C01822=1228.757,-113.151,-35.858,179.412,5.295,149.097
C01823=1228.752,-112.901,-35.869,179.414,5.294,149.096
C01824=1228.747,-112.651,-35.879,179.416,5.295,149.096
C01825=1228.741,-112.401,-35.889,179.418,5.294,149.095
C01826=1228.736,-112.152,-35.899,179.421,5.295,149.094
C01827=1228.731,-111.902,-35.910,179.423,5.295,149.094
C01828=1228.726,-111.652,-35.920,179.425,5.295,149.093
C01829=1228.720,-111.403,-35.930,179.427,5.295,149.092
C01830=1228.715,-111.153,-35.941,179.430,5.295,149.091
C01831=1228.710,-110.903,-35.950,179.432,5.295,149.091
C01832=1228.704,-110.653,-35.960,179.434,5.295,149.090
C01833=1228.699,-110.403,-35.970,179.437,5.295,149.089
C01834=1228.694,-110.153,-35.980,179.439,5.295,149.089
C01835=1228.688,-109.904,-35.991,179.442,5.295,149.088
C01836=1228.684,-109.655,-36.001,179.443,5.295,149.087
C01837=1228.679,-109.405,-36.012,179.446,5.296,149.087
C01838=1228.673,-109.156,-36.022,179.448,5.295,149.086
C01839=1228.668,-108.905,-36.032,179.451,5.296,149.085
C01840=1228.662,-108.656,-36.043,179.453,5.295,149.085
C01841=1228.657,-108.405,-36.053,179.456,5.296,149.084
C01842=1228.653,-108.156,-36.063,179.458,5.295,149.083
C01843=1228.647,-107.907,-36.073,179.460,5.296,149.082
C01844=1228.642,-107.656,-36.084,179.462,5.295,149.082
C01845=1228.636,-107.407,-36.094,179.465,5.296,149.081
C01846=1228.631,-107.157,-36.104,179.467,5.296,149.080
C01847=1228.626,-106.907,-36.115,179.469,5.295,149.080
C01848=1228.621,-106.658,-36.124,179.471,5.296,149.079
C01849=1228.616,-106.408,-36.135,179.474,5.296,149.078
C01850=1228.610,-106.158,-36.145,179.476,5.296,149.078
C01851=1228.606,-105.908,-36.156,179.478,5.296,149.077
C01852=1228.600,-105.659,-36.166,179.481,5.296,149.076
C01853=1228.595,-105.409,-36.177,179.483,5.296,149.075
C01854=1228.589,-105.159,-36.187,179.486,5.296,149.075
C01855=1228.584,-104.910,-36.197,179.488,5.296,149.074
C01856=1228.579,-104.659,-36.208,179.491,5.296,149.073
C01857=1228.574,-104.410,-36.218,179.492,5.296,149.073
C01858=1228.569,-104.160,-36.228,179.495,5.297,149.072
C01859=1228.564,-103.911,-36.239,179.497,5.296,149.071
C01860=1228.559,-103.661,-36.250,179.500,5.297,149.071
C01861=1228.553,-103.411,-36.260,179.502,5.296,149.070
C01862=1228.548,-103.161,-36.270,179.504,5.296,149.069
C01863=1228.542,-102.911,-36.281,179.506,5.296,149.069
C01864=1228.537,-102.662,-36.292,179.509,5.296,149.068
C01865=1228.532,-102.412,-36.302,179.511,5.296,149.067
C01866=1228.527,-102.163,-36.312,179.513,5.296,149.066
C01867=1228.522,-101.912,-36.323,179.516,5.297,149.066
C01868=1228.516,-101.663,-36.333,179.518,5.296,149.065
C01869=1228.511,-101.413,-36.344,179.521,5.297,149.064
C01870=1228.506,-101.164,-36.355,179.522,5.297,149.064
C01871=1228.501,-100.892,-36.366,179.526,5.297,149.063
C01872=1228.495,-100.621,-36.378,179.528,5.296,149.062
C01873=1228.489,-100.351,-36.388,179.530,5.297,149.061
C01874=1228.483,-100.080,-36.401,179.533,5.297,149.061
C01875=1228.478,-99.830,-36.411,179.535,5.297,149.060
C01876=1228.473,-99.580,-36.421,179.538,5.297,149.059
C01877=1228.468,-99.330,-36.433,179.540,5.297,149.059
C01878=1228.463,-99.081,-36.443,179.543,5.297,149.058
C01879=1228.458,-98.831,-36.454,179.545,5.297,149.057
C01880=1228.452,-98.581,-36.464,179.547,5.297,149.056
C01881=1228.447,-98.332,-36.475,179.549,5.297,149.056
C01882=1228.442,-98.082,-36.485,179.552,5.298,149.055
C01883=1228.437,-97.832,-36.496,179.554,5.297,149.054
C01884=1228.431,-97.583,-36.507,179.556,5.297,149.054
C01885=1228.426,-97.333,-36.517,179.558,5.298,149.053
C01886=1228.421,-97.083,-36.528,179.561,5.297,149.052
C01887=1228.416,-96.833,-36.539,179.563,5.298,149.052
C01888=1228.411,-96.584,-36.549,179.565,5.297,149.051
C01889=1228.406,-96.334,-36.560,179.568,5.298,149.050
C01890=1228.400,-96.084,-36.571,179.570,5.297,149.050
C01891=1228.395,-95.834,-36.582,179.573,5.298,149.049
C01892=1228.390,-95.584,-36.593,179.575,5.298,149.048
C01893=1228.384,-95.335,-36.603,179.578,5.298,149.047
C01894=1228.380,-95.085,-36.615,179.580,5.298,149.047
C01895=1228.374,-94.836,-36.625,179.582,5.298,149.046
C01896=1228.369,-94.586,-36.635,179.584,5.298,149.045
C01897=1228.364,-94.337,-36.646,179.587,5.298,149.045
C01898=1228.359,-94.086,-36.657,179.589,5.298,149.044
C01899=1228.353,-93.837,-36.668,179.592,5.298,149.043
C01900=1228.348,-93.587,-36.679,179.593,5.298,149.043
C01901=1228.343,-93.337,-36.690,179.596,5.299,149.042
C01902=1228.337,-93.088,-36.700,179.598,5.298,149.041
C01903=1228.333,-92.838,-36.712,179.601,5.299,149.041
C01904=1228.327,-92.589,-36.722,179.603,5.298,149.040
C01905=1228.322,-92.338,-36.732,179.606,5.299,149.039
C01906=1228.317,-92.089,-36.744,179.608,5.299,149.038
C01907=1228.311,-91.839,-36.755,179.610,5.299,149.038
C01908=1228.306,-91.589,-36.766,179.612,5.299,149.037
C01909=1228.301,-91.340,-36.776,179.615,5.299,149.036
C01910=1228.296,-91.090,-36.787,179.617,5.299,149.036
C01911=1228.291,-90.840,-36.799,179.620,5.299,149.035
C01912=1228.285,-90.591,-36.809,179.622,5.299,149.034
C01913=1228.280,-90.341,-36.821,179.625,5.299,149.033
C01914=1228.275,-90.091,-36.831,179.627,5.299,149.033
C01915=1228.270,-89.842,-36.842,179.629,5.299,149.032
C01916=1228.265,-89.592,-36.853,179.632,5.299,149.031
C01917=1228.259,-89.342,-36.864,179.634,5.299,149.031
C01918=1228.254,-89.092,-36.875,179.636,5.299,149.030
C01919=1228.249,-88.842,-36.886,179.639,5.299,149.029
C01920=1228.244,-88.593,-36.897,179.641,5.299,149.028
C01921=1228.239,-88.343,-36.908,179.643,5.300,149.028
C01922=1228.234,-88.093,-36.920,179.645,5.300,149.027
C01923=1228.228,-87.844,-36.930,179.648,5.300,149.027
C01924=1228.223,-87.594,-36.941,179.650,5.300,149.026
C01925=1228.219,-87.345,-36.952,179.653,5.300,149.025
C01926=1228.212,-87.095,-36.963,179.655,5.300,149.024
C01927=1228.208,-86.845,-36.974,179.658,5.300,149.024
C01928=1228.203,-86.595,-36.985,179.660,5.300,149.023
C01929=1228.197,-86.346,-36.996,179.662,5.300,149.022
C01930=1228.192,-86.096,-37.008,179.664,5.300,149.022
C01931=1228.187,-85.846,-37.018,179.667,5.300,149.021
C01932=1228.182,-85.597,-37.029,179.669,5.300,149.020
C01933=1228.177,-85.347,-37.041,179.672,5.301,149.019
C01934=1228.171,-85.097,-37.052,179.674,5.300,149.019
C01935=1228.166,-84.848,-37.063,179.677,5.301,149.018
C01936=1228.161,-84.598,-37.074,179.679,5.300,149.017
C01937=1228.156,-84.348,-37.086,179.681,5.301,149.017
C01938=1228.151,-84.098,-37.096,179.683,5.300,149.016
C01939=1228.145,-83.849,-37.107,179.686,5.301,149.015
C01940=1228.140,-83.599,-37.119,179.688,5.300,149.014
C01941=1228.135,-83.349,-37.130,179.691,5.301,149.014
C01942=1228.130,-83.100,-37.141,179.693,5.301,149.013
C01943=1228.124,-82.850,-37.153,179.696,5.301,149.012
C01944=1228.120,-82.600,-37.164,179.698,5.301,149.012
C01945=1228.115,-82.350,-37.175,179.700,5.301,149.011
C01946=1228.109,-82.101,-37.186,179.702,5.301,149.010
C01947=1228.104,-81.851,-37.197,179.705,5.301,149.009
C01948=1228.099,-81.602,-37.209,179.707,5.301,149.009
C01949=1228.094,-81.352,-37.221,179.710,5.301,149.008
C01950=1228.088,-81.102,-37.231,179.712,5.301,149.007
C01951=1228.083,-80.852,-37.242,179.714,5.302,149.007
C01952=1228.078,-80.602,-37.254,179.716,5.301,149.006
C01953=1228.073,-80.353,-37.265,179.719,5.302,149.005
C01954=1228.067,-80.104,-37.277,179.721,5.302,149.005
C01955=1228.062,-79.853,-37.287,179.724,5.302,149.004
C01956=1228.058,-79.604,-37.299,179.726,5.302,149.003
C01957=1228.052,-79.354,-37.310,179.728,5.302,149.003
C01958=1228.047,-79.105,-37.321,179.731,5.302,149.002
C01959=1228.041,-78.855,-37.333,179.733,5.302,149.001
C01960=1228.037,-78.605,-37.345,179.735,5.302,149.000
C01961=1228.032,-78.356,-37.356,179.738,5.302,149.000
C01962=1228.026,-78.105,-37.367,179.740,5.302,148.999
C01963=1228.021,-77.856,-37.378,179.743,5.302,148.998
C01964=1228.016,-77.606,-37.390,179.745,5.302,148.998
C01965=1228.011,-77.357,-37.401,179.748,5.303,148.997
C01966=1228.006,-77.107,-37.413,179.750,5.302,148.996
C01967=1228.001,-76.857,-37.424,179.752,5.303,148.996
C01968=1227.995,-76.608,-37.436,179.754,5.302,148.995
C01969=1227.990,-76.358,-37.447,179.757,5.303,148.994
C01970=1227.985,-76.108,-37.459,179.759,5.302,148.993
C01971=1227.980,-75.859,-37.470,179.762,5.303,148.993
C01972=1227.975,-75.609,-37.482,179.764,5.303,148.992
C01973=1227.969,-75.359,-37.492,179.767,5.303,148.991
C01974=1227.964,-75.109,-37.504,179.769,5.304,148.991
C01975=1227.959,-74.839,-37.517,179.771,5.303,148.990
C01976=1227.953,-74.570,-37.529,179.774,5.304,148.989
C01977=1227.947,-74.299,-37.541,179.777,5.304,148.988
C01978=1227.942,-74.028,-37.554,179.779,5.303,148.987
C01979=1227.937,-73.778,-37.566,179.782,5.304,148.987
C01980=1227.931,-73.529,-37.577,179.784,5.303,148.986
C01981=1227.926,-73.279,-37.589,179.787,5.304,148.985
C01982=1227.921,-73.030,-37.600,179.789,5.304,148.985
C01983=1227.916,-72.780,-37.612,179.791,5.304,148.984
C01984=1227.911,-72.530,-37.624,179.794,5.304,148.983
C01985=1227.906,-72.280,-37.635,179.796,5.304,148.983
C01986=1227.900,-72.030,-37.647,179.798,5.304,148.982
C01987=1227.895,-71.781,-37.658,179.801,5.304,148.981
C01988=1227.890,-71.531,-37.670,179.803,5.304,148.980
C01989=1227.885,-71.282,-37.681,179.806,5.304,148.980
C01990=1227.879,-71.032,-37.693,179.808,5.304,148.979
C01991=1227.875,-70.782,-37.705,179.810,5.305,148.978
C01992=1227.869,-70.532,-37.717,179.813,5.305,148.978
C01993=1227.864,-70.282,-37.728,179.815,5.305,148.977
C01994=1227.859,-70.033,-37.740,179.818,5.305,148.976
C01995=1227.853,-69.784,-37.752,179.820,5.305,148.975
C01996=1227.849,-69.535,-37.763,179.823,5.305,148.975
C01997=1227.843,-69.285,-37.775,179.825,5.305,148.974
C01998=1227.838,-69.035,-37.787,179.827,5.305,148.973
C01999=1227.833,-68.785,-37.798,179.830,5.305,148.973
C02000=1227.828,-68.535,-37.810,179.832,5.305,148.972
C02001=1227.822,-68.285,-37.822,179.834,5.305,148.971
C02002=1227.818,-68.036,-37.833,179.837,5.306,148.971
C02003=1227.813,-67.786,-37.846,179.839,5.305,148.970
C02004=1227.807,-67.536,-37.858,179.842,5.306,148.969
C02005=1227.802,-67.287,-37.869,179.844,5.306,148.968
C02006=1227.797,-67.037,-37.881,179.846,5.306,148.968
C02007=1227.791,-66.788,-37.893,179.849,5.306,148.967
C02008=1227.787,-66.539,-37.905,179.851,5.306,148.966
C02009=1227.781,-66.289,-37.916,179.854,5.306,148.966
C02010=1227.776,-66.039,-37.928,179.856,5.306,148.965
C02011=1227.771,-65.789,-37.940,179.859,5.307,148.964
C02012=1227.766,-65.539,-37.951,179.861,5.306,148.963
C02013=1227.760,-65.290,-37.964,179.863,5.307,148.963
C02014=1227.756,-65.040,-37.975,179.866,5.306,148.962
C02015=1227.750,-64.790,-37.987,179.868,5.307,148.961
C02016=1227.745,-64.540,-37.999,179.870,5.307,148.961
C02017=1227.741,-64.291,-38.011,179.873,5.307,148.960
C02018=1227.735,-64.041,-38.023,179.876,5.307,148.959
C02019=1227.730,-63.791,-38.035,179.878,5.307,148.958
C02020=1227.725,-63.542,-38.048,179.880,5.308,148.958
C02021=1227.720,-63.292,-38.059,179.882,5.307,148.957
C02022=1227.714,-63.042,-38.071,179.885,5.308,148.956
C02023=1227.709,-62.793,-38.083,179.887,5.307,148.956
C02024=1227.704,-62.543,-38.095,179.890,5.308,148.955
C02025=1227.699,-62.294,-38.106,179.892,5.307,148.954
C02026=1227.694,-62.044,-38.118,179.895,5.308,148.954
C02027=1227.689,-61.794,-38.131,179.897,5.308,148.953
C02028=1227.683,-61.544,-38.143,179.899,5.308,148.952
C02029=1227.679,-61.295,-38.154,179.902,5.309,148.951
C02030=1227.673,-61.045,-38.167,179.904,5.308,148.951
C02031=1227.668,-60.796,-38.179,179.907,5.309,148.950
C02032=1227.663,-60.546,-38.191,179.909,5.308,148.949
C02033=1227.658,-60.297,-38.203,179.912,5.309,148.949
C02034=1227.653,-60.047,-38.214,179.914,5.309,148.948
C02035=1227.648,-59.797,-38.227,179.916,5.309,148.947
C02036=1227.642,-59.547,-38.239,179.919,5.309,148.947
C02037=1227.637,-59.298,-38.251,179.921,5.309,148.946
C02038=1227.632,-59.048,-38.263,179.924,5.310,148.945
C02039=1227.627,-58.799,-38.275,179.926,5.309,148.944
C02040=1227.622,-58.549,-38.287,179.928,5.310,148.944
C02041=1227.616,-58.299,-38.299,179.931,5.309,148.943
C02042=1227.612,-58.049,-38.312,179.933,5.310,148.942
C02043=1227.606,-57.799,-38.324,179.935,5.310,148.942
C02044=1227.602,-57.550,-38.336,179.938,5.310,148.941
C02045=1227.597,-57.300,-38.348,179.941,5.310,148.940
C02046=1227.591,-57.051,-38.360,179.943,5.310,148.939
C02047=1227.586,-56.801,-38.372,179.945,5.311,148.939
C02048=1227.581,-56.551,-38.384,179.948,5.310,148.938
C02049=1227.576,-56.302,-38.397,179.950,5.311,148.937
C02050=1227.570,-56.052,-38.409,179.952,5.310,148.937
C02051=1227.566,-55.803,-38.421,179.955,5.311,148.936
C02052=1227.561,-55.554,-38.433,179.958,5.311,148.935
C02053=1227.555,-55.304,-38.445,179.960,5.311,148.935
C02054=1227.551,-55.054,-38.458,179.962,5.312,148.934
C02055=1227.545,-54.804,-38.470,179.964,5.311,148.933
C02056=1227.540,-54.554,-38.483,179.967,5.312,148.932
C02057=1227.535,-54.304,-38.495,179.969,5.311,148.932
C02058=1227.530,-54.055,-38.507,179.972,5.312,148.931
C02059=1227.524,-53.805,-38.519,179.975,5.312,148.930
C02060=1227.519,-53.556,-38.532,179.977,5.312,148.930
C02061=1227.514,-53.306,-38.544,179.979,5.312,148.929
C02062=1227.509,-53.057,-38.556,179.981,5.312,148.928
C02063=1227.505,-52.807,-38.569,179.984,5.313,148.927
C02064=1227.499,-52.557,-38.580,179.986,5.312,148.927
C02065=1227.494,-52.308,-38.593,179.989,5.313,148.926
C02066=1227.489,-52.058,-38.605,179.991,5.313,148.925
C02067=1227.484,-51.808,-38.617,179.994,5.313,148.925
C02068=1227.478,-51.559,-38.630,179.996,5.313,148.924
C02069=1227.473,-51.309,-38.642,179.998,5.313,148.923
C02070=1227.468,-51.059,-38.655,-179.999,5.314,148.923
C02071=1227.463,-50.810,-38.668,-179.997,5.313,148.922
C02072=1227.458,-50.560,-38.679,-179.994,5.314,148.921
C02073=1227.453,-50.311,-38.692,-179.992,5.314,148.920
C02074=1227.448,-50.061,-38.705,-179.990,5.314,148.920
C02075=1227.442,-49.811,-38.717,-179.987,5.314,148.919
C02076=1227.438,-49.561,-38.729,-179.985,5.314,148.918
C02077=1227.433,-49.312,-38.742,-179.982,5.314,148.918
C02078=1227.427,-49.062,-38.754,-179.980,5.314,148.917
C02079=1227.421,-48.792,-38.768,-179.977,5.315,148.916
C02080=1227.416,-48.523,-38.782,-179.974,5.315,148.915
C02081=1227.410,-48.253,-38.795,-179.972,5.315,148.915
C02082=1227.405,-47.983,-38.808,-179.969,5.315,148.914
C02083=1227.400,-47.733,-38.821,-179.967,5.315,148.913
C02084=1227.394,-47.484,-38.834,-179.964,5.316,148.912
C02085=1227.389,-47.234,-38.846,-179.962,5.316,148.912
C02086=1227.384,-46.985,-38.858,-179.959,5.316,148.911
C02087=1227.379,-46.735,-38.871,-179.957,5.316,148.910
C02088=1227.374,-46.485,-38.884,-179.955,5.316,148.910
C02089=1227.369,-46.235,-38.896,-179.953,5.316,148.909
C02090=1227.364,-45.986,-38.909,-179.950,5.316,148.908
C02091=1227.359,-45.736,-38.922,-179.947,5.317,148.908
C02092=1227.354,-45.487,-38.934,-179.945,5.316,148.907
C02093=1227.349,-45.237,-38.947,-179.942,5.317,148.906
C02094=1227.344,-44.988,-38.959,-179.940,5.317,148.905
C02095=1227.338,-44.738,-38.972,-179.938,5.317,148.905
C02096=1227.333,-44.488,-38.985,-179.935,5.318,148.904
C02097=1227.328,-44.239,-38.997,-179.933,5.317,148.903
C02098=1227.323,-43.989,-39.010,-179.930,5.317,148.902
C02099=1227.318,-43.740,-39.023,-179.928,5.317,148.902
C02100=1227.313,-43.490,-39.036,-179.925,5.318,148.901
C02101=1227.308,-43.240,-39.047,-179.922,5.318,148.900
C02102=1227.302,-42.990,-39.061,-179.920,5.318,148.900
C02103=1227.297,-42.741,-39.073,-179.918,5.318,148.899
C02104=1227.292,-42.491,-39.086,-179.916,5.318,148.898
C02105=1227.287,-42.242,-39.099,-179.913,5.318,148.898
C02106=1227.282,-41.992,-39.111,-179.910,5.319,148.897
C02107=1227.278,-41.742,-39.124,-179.908,5.319,148.896
C02108=1227.272,-41.493,-39.138,-179.905,5.319,148.895
C02109=1227.267,-41.243,-39.150,-179.903,5.319,148.895
C02110=1227.261,-40.994,-39.163,-179.901,5.319,148.894
C02111=1227.257,-40.744,-39.176,-179.898,5.320,148.893
C02112=1227.251,-40.494,-39.188,-179.896,5.319,148.893
C02113=1227.246,-40.245,-39.200,-179.893,5.320,148.892
C02114=1227.241,-39.994,-39.214,-179.891,5.320,148.891
C02115=1227.236,-39.745,-39.226,-179.889,5.320,148.891
C02116=1227.231,-39.496,-39.239,-179.886,5.321,148.890
C02117=1227.226,-39.246,-39.252,-179.884,5.320,148.889
C02118=1227.220,-38.996,-39.265,-179.881,5.321,148.888
C02119=1227.215,-38.747,-39.278,-179.878,5.321,148.888
C02120=1227.211,-38.497,-39.291,-179.876,5.321,148.887
C02121=1227.206,-38.248,-39.303,-179.874,5.321,148.886
C02122=1227.200,-37.998,-39.316,-179.872,5.321,148.886
C02123=1227.195,-37.748,-39.329,-179.869,5.322,148.885
C02124=1227.190,-37.499,-39.342,-179.866,5.322,148.884
C02125=1227.185,-37.249,-39.355,-179.864,5.322,148.884
C02126=1227.180,-37.000,-39.369,-179.862,5.322,148.883
C02127=1227.175,-36.750,-39.382,-179.860,5.322,148.882
C02128=1227.170,-36.501,-39.394,-179.857,5.322,148.881
C02129=1227.165,-36.251,-39.408,-179.854,5.323,148.881
C02130=1227.159,-36.001,-39.420,-179.852,5.323,148.880
C02131=1227.154,-35.752,-39.433,-179.849,5.323,148.879
C02132=1227.149,-35.502,-39.446,-179.847,5.324,148.879
C02133=1227.144,-35.252,-39.459,-179.845,5.323,148.878
C02134=1227.139,-35.003,-39.472,-179.842,5.324,148.877
C02135=1227.134,-34.753,-39.485,-179.840,5.323,148.877
C02136=1227.128,-34.503,-39.498,-179.837,5.324,148.876
C02137=1227.124,-34.254,-39.511,-179.835,5.324,148.875
C02138=1227.119,-34.005,-39.524,-179.833,5.324,148.874
C02139=1227.113,-33.755,-39.537,-179.830,5.325,148.874
C02140=1227.109,-33.505,-39.550,-179.827,5.325,148.873
C02141=1227.103,-33.255,-39.563,-179.825,5.325,148.872
C02142=1227.098,-33.005,-39.576,-179.822,5.325,148.872
C02143=1227.094,-32.757,-39.590,-179.820,5.325,148.871
C02144=1227.088,-32.507,-39.603,-179.818,5.325,148.870
C02145=1227.083,-32.257,-39.616,-179.815,5.326,148.870
C02146=1227.078,-32.008,-39.629,-179.813,5.326,148.869
C02147=1227.073,-31.757,-39.642,-179.810,5.326,148.868
C02148=1227.068,-31.509,-39.655,-179.808,5.327,148.867
C02149=1227.062,-31.259,-39.669,-179.806,5.326,148.867
C02150=1227.058,-31.009,-39.682,-179.803,5.327,148.866
C02151=1227.052,-30.760,-39.694,-179.801,5.326,148.865
C02152=1227.047,-30.510,-39.708,-179.798,5.327,148.865
C02153=1227.042,-30.261,-39.721,-179.796,5.327,148.864
C02154=1227.037,-30.010,-39.735,-179.793,5.327,148.863
C02155=1227.032,-29.761,-39.747,-179.791,5.328,148.863
C02156=1227.027,-29.511,-39.761,-179.788,5.328,148.862
C02157=1227.022,-29.262,-39.774,-179.786,5.327,148.861
C02158=1227.017,-29.013,-39.787,-179.783,5.328,148.860
C02159=1227.012,-28.762,-39.800,-179.780,5.328,148.860
C02160=1227.007,-28.514,-39.814,-179.778,5.328,148.859
C02161=1227.001,-28.263,-39.827,-179.775,5.329,148.858
C02162=1226.996,-28.014,-39.840,-179.773,5.329,148.857
C02163=1226.991,-27.764,-39.854,-179.771,5.329,148.857
C02164=1226.986,-27.515,-39.867,-179.768,5.329,148.856
C02165=1226.981,-27.265,-39.880,-179.766,5.329,148.855
C02166=1226.976,-27.016,-39.893,-179.763,5.329,148.855
C02167=1226.971,-26.766,-39.907,-179.761,5.330,148.854
C02168=1226.966,-26.516,-39.920,-179.759,5.330,148.853
C02169=1226.961,-26.267,-39.934,-179.756,5.330,148.853
C02170=1226.956,-26.017,-39.946,-179.753,5.331,148.852
C02171=1226.951,-25.768,-39.961,-179.751,5.330,148.851
C02172=1226.946,-25.518,-39.973,-179.749,5.331,148.850
C02173=1226.940,-25.268,-39.987,-179.746,5.331,148.850
C02174=1226.936,-25.019,-40.000,-179.744,5.331,148.849
C02175=1226.930,-24.769,-40.014,-179.741,5.332,148.848
C02176=1226.925,-24.520,-40.027,-179.738,5.332,148.848
C02177=1226.920,-24.270,-40.041,-179.736,5.332,148.847
C02178=1226.915,-24.021,-40.054,-179.734,5.332,148.846
C02179=1226.910,-23.771,-40.068,-179.731,5.333,148.846
C02180=1226.905,-23.521,-40.080,-179.729,5.332,148.845
C02181=1226.900,-23.272,-40.094,-179.726,5.333,148.844
C02182=1226.895,-23.021,-40.108,-179.724,5.333,148.843
C02183=1226.889,-22.753,-40.122,-179.722,5.333,148.843
C02184=1226.884,-22.484,-40.137,-179.719,5.334,148.842
C02185=1226.879,-22.214,-40.152,-179.716,5.334,148.841
C02186=1226.873,-21.944,-40.166,-179.713,5.334,148.840
C02187=1226.868,-21.695,-40.180,-179.711,5.334,148.840
C02188=1226.863,-21.445,-40.193,-179.708,5.334,148.839
C02189=1226.858,-21.196,-40.206,-179.706,5.335,148.838
C02190=1226.853,-20.946,-40.220,-179.704,5.335,148.838
C02191=1226.847,-20.697,-40.234,-179.701,5.335,148.837
C02192=1226.843,-20.448,-40.248,-179.698,5.336,148.836
C02193=1226.837,-20.198,-40.261,-179.696,5.335,148.836
C02194=1226.832,-19.948,-40.275,-179.694,5.336,148.835
C02195=1226.828,-19.698,-40.288,-179.691,5.336,148.834
C02196=1226.822,-19.449,-40.302,-179.689,5.336,148.834
C02197=1226.817,-19.199,-40.316,-179.686,5.337,148.833
C02198=1226.812,-18.950,-40.329,-179.683,5.337,148.832
C02199=1226.807,-18.701,-40.343,-179.681,5.337,148.831
C02200=1226.802,-18.450,-40.357,-179.679,5.337,148.831
C02201=1226.797,-18.202,-40.370,-179.676,5.338,148.830
C02202=1226.792,-17.951,-40.384,-179.674,5.338,148.829
C02203=1226.786,-17.702,-40.398,-179.671,5.338,148.829
C02204=1226.782,-17.453,-40.411,-179.669,5.339,148.828
C02205=1226.777,-17.203,-40.425,-179.667,5.338,148.827
C02206=1226.771,-16.954,-40.439,-179.664,5.339,148.827
C02207=1226.767,-16.704,-40.452,-179.661,5.339,148.826
C02208=1226.762,-16.454,-40.466,-179.659,5.339,148.825
C02209=1226.756,-16.205,-40.480,-179.657,5.339,148.824
C02210=1226.751,-15.955,-40.494,-179.654,5.340,148.824
C02211=1226.747,-15.705,-40.507,-179.651,5.340,148.823
C02212=1226.741,-15.456,-40.521,-179.649,5.340,148.822
C02213=1226.736,-15.206,-40.535,-179.647,5.341,148.822
C02214=1226.730,-14.957,-40.548,-179.644,5.341,148.821
C02215=1226.726,-14.707,-40.562,-179.642,5.341,148.820
C02216=1226.721,-14.458,-40.576,-179.639,5.341,148.820
C02217=1226.715,-14.209,-40.590,-179.636,5.342,148.819
C02218=1226.710,-13.958,-40.604,-179.634,5.342,148.818
C02219=1226.706,-13.709,-40.618,-179.632,5.342,148.818
C02220=1226.700,-13.460,-40.631,-179.629,5.343,148.817
C02221=1226.695,-13.210,-40.646,-179.627,5.342,148.816
C02222=1226.690,-12.960,-40.659,-179.624,5.343,148.815
C02223=1226.686,-12.710,-40.673,-179.622,5.343,148.815
C02224=1226.680,-12.461,-40.687,-179.620,5.343,148.814
C02225=1226.676,-12.212,-40.701,-179.617,5.344,148.813
C02226=1226.671,-11.962,-40.715,-179.614,5.344,148.813
C02227=1226.665,-11.712,-40.729,-179.612,5.345,148.812
C02228=1226.660,-11.463,-40.743,-179.610,5.344,148.811
C02229=1226.656,-11.213,-40.757,-179.607,5.345,148.811
C02230=1226.650,-10.964,-40.771,-179.604,5.345,148.810
C02231=1226.645,-10.714,-40.785,-179.602,5.345,148.809
C02232=1226.640,-10.465,-40.799,-179.600,5.346,148.809
C02233=1226.635,-10.214,-40.813,-179.597,5.346,148.808
C02234=1226.629,-9.965,-40.827,-179.595,5.346,148.807
C02235=1226.625,-9.716,-40.840,-179.592,5.346,148.806
C02236=1226.620,-9.466,-40.855,-179.589,5.347,148.806
C02237=1226.615,-9.217,-40.869,-179.587,5.347,148.805
C02238=1226.610,-8.968,-40.883,-179.585,5.347,148.804
C02239=1226.605,-8.718,-40.897,-179.582,5.348,148.804
C02240=1226.600,-8.468,-40.911,-179.579,5.348,148.803
C02241=1226.595,-8.218,-40.926,-179.577,5.348,148.802
C02242=1226.589,-7.969,-40.939,-179.575,5.348,148.802
C02243=1226.585,-7.719,-40.952,-179.572,5.349,148.801
C02244=1226.580,-7.470,-40.967,-179.569,5.349,148.800
C02245=1226.575,-7.220,-40.981,-179.567,5.349,148.800
C02246=1226.569,-6.971,-40.995,-179.565,5.349,148.799
C02247=1226.564,-6.721,-41.009,-179.562,5.350,148.798
C02248=1226.559,-6.472,-41.023,-179.560,5.350,148.797
C02249=1226.554,-6.222,-41.038,-179.557,5.350,148.797
C02250=1226.549,-5.972,-41.052,-179.555,5.351,148.796
C02251=1226.544,-5.723,-41.066,-179.552,5.351,148.795
C02252=1226.539,-5.473,-41.080,-179.550,5.351,148.795
C02253=1226.534,-5.224,-41.094,-179.547,5.351,148.794
C02254=1226.529,-4.974,-41.109,-179.545,5.352,148.793
C02255=1226.523,-4.725,-41.123,-179.542,5.352,148.793
C02256=1226.518,-4.475,-41.137,-179.540,5.352,148.792
C02257=1226.513,-4.226,-41.151,-179.537,5.353,148.791
C02258=1226.508,-3.976,-41.165,-179.535,5.353,148.791
C02259=1226.504,-3.726,-41.180,-179.532,5.353,148.790
C02260=1226.499,-3.477,-41.195,-179.530,5.353,148.789
C02261=1226.493,-3.228,-41.209,-179.527,5.354,148.789
C02262=1226.488,-2.978,-41.223,-179.525,5.354,148.788
C02263=1226.483,-2.729,-41.237,-179.522,5.354,148.787
C02264=1226.478,-2.479,-41.251,-179.520,5.355,148.786
C02265=1226.474,-2.229,-41.266,-179.517,5.355,148.786
C02266=1226.469,-1.980,-41.280,-179.515,5.355,148.785
C02267=1226.463,-1.731,-41.294,-179.512,5.356,148.784
C02268=1226.458,-1.481,-41.308,-179.510,5.356,148.784
C02269=1226.453,-1.231,-41.323,-179.507,5.357,148.783
C02270=1226.448,-0.982,-41.337,-179.505,5.356,148.782
C02271=1226.443,-0.732,-41.352,-179.502,5.357,148.782
C02272=1226.439,-0.483,-41.366,-179.500,5.357,148.781
C02273=1226.434,-0.233,-41.380,-179.497,5.358,148.780
C02274=1226.428,0.016,-41.394,-179.495,5.358,148.780
C02275=1226.423,0.266,-41.409,-179.492,5.358,148.779
C02276=1226.418,0.515,-41.424,-179.490,5.359,148.778
C02277=1226.413,0.765,-41.438,-179.488,5.358,148.777
C02278=1226.409,1.014,-41.452,-179.485,5.359,148.777
C02279=1226.403,1.264,-41.467,-179.482,5.359,148.776
C02280=1226.398,1.514,-41.481,-179.480,5.360,148.775
C02281=1226.393,1.763,-41.496,-179.478,5.360,148.775
C02282=1226.388,2.012,-41.510,-179.475,5.360,148.774
C02283=1226.383,2.262,-41.524,-179.472,5.361,148.773
C02284=1226.378,2.512,-41.539,-179.470,5.361,148.773
C02285=1226.373,2.761,-41.554,-179.467,5.361,148.772
C02286=1226.368,3.010,-41.568,-179.465,5.361,148.771
C02287=1226.362,3.280,-41.584,-179.462,5.362,148.771
C02288=1226.357,3.548,-41.600,-179.460,5.362,148.770
C02289=1226.352,3.818,-41.615,-179.456,5.363,148.769
C02290=1226.347,4.087,-41.631,-179.454,5.363,148.768
C02291=1226.342,4.336,-41.645,-179.451,5.364,148.768
C02292=1226.336,4.586,-41.661,-179.449,5.363,148.767
C02293=1226.331,4.835,-41.675,-179.446,5.364,148.766
C02294=1226.326,5.084,-41.689,-179.444,5.364,148.766
C02295=1226.321,5.333,-41.704,-179.441,5.365,148.765
C02296=1226.316,5.583,-41.718,-179.439,5.365,148.764
C02297=1226.310,5.833,-41.733,-179.436,5.365,148.763
C02298=1226.306,6.082,-41.748,-179.434,5.366,148.763
C02299=1226.301,6.332,-41.762,-179.431,5.366,148.762
C02300=1226.296,6.581,-41.777,-179.429,5.366,148.761
C02301=1226.291,6.831,-41.791,-179.426,5.366,148.761
C02302=1226.286,7.081,-41.806,-179.424,5.367,148.760
C02303=1226.281,7.330,-41.821,-179.421,5.368,148.759
C02304=1226.276,7.580,-41.836,-179.419,5.367,148.759
C02305=1226.271,7.829,-41.851,-179.416,5.368,148.758
C02306=1226.266,8.079,-41.865,-179.414,5.368,148.757
C02307=1226.261,8.328,-41.880,-179.411,5.369,148.757
C02308=1226.256,8.577,-41.895,-179.409,5.369,148.756
C02309=1226.251,8.827,-41.909,-179.407,5.369,148.755
C02310=1226.246,9.077,-41.925,-179.404,5.370,148.755
C02311=1226.241,9.326,-41.939,-179.401,5.371,148.754
C02312=1226.236,9.575,-41.954,-179.399,5.371,148.753
C02313=1226.230,9.825,-41.969,-179.397,5.371,148.753
C02314=1226.226,10.075,-41.984,-179.394,5.371,148.752
C02315=1226.221,10.324,-41.998,-179.391,5.372,148.751
C02316=1226.216,10.573,-42.013,-179.389,5.372,148.751
C02317=1226.210,10.823,-42.028,-179.387,5.372,148.750
C02318=1226.206,11.072,-42.043,-179.384,5.373,148.749
C02319=1226.201,11.322,-42.057,-179.381,5.373,148.749
C02320=1226.195,11.572,-42.073,-179.379,5.374,148.748
C02321=1226.190,11.821,-42.087,-179.376,5.374,148.747
C02322=1226.186,12.070,-42.102,-179.374,5.374,148.747
C02323=1226.180,12.320,-42.117,-179.371,5.374,148.746
C02324=1226.175,12.569,-42.132,-179.369,5.375,148.745
C02325=1226.171,12.819,-42.147,-179.366,5.376,148.745
C02326=1226.166,13.069,-42.162,-179.364,5.375,148.744
C02327=1226.161,13.318,-42.177,-179.361,5.376,148.743
C02328=1226.155,13.568,-42.192,-179.359,5.376,148.742
C02329=1226.151,13.817,-42.207,-179.356,5.377,148.742
C02330=1226.146,14.067,-42.222,-179.353,5.377,148.741
C02331=1226.140,14.317,-42.237,-179.351,5.377,148.740
C02332=1226.136,14.566,-42.252,-179.349,5.378,148.740
C02333=1226.131,14.815,-42.266,-179.346,5.378,148.739
C02334=1226.125,15.065,-42.282,-179.343,5.379,148.738
C02335=1226.121,15.314,-42.297,-179.341,5.379,148.738
C02336=1226.115,15.564,-42.311,-179.339,5.379,148.737
C02337=1226.110,15.813,-42.326,-179.336,5.380,148.736
C02338=1226.106,16.063,-42.342,-179.333,5.380,148.736
C02339=1226.101,16.313,-42.357,-179.331,5.381,148.735
C02340=1226.096,16.562,-42.372,-179.329,5.381,148.734
C02341=1226.091,16.811,-42.387,-179.326,5.381,148.734
C02342=1226.086,17.060,-42.402,-179.324,5.382,148.733
C02343=1226.080,17.310,-42.417,-179.321,5.382,148.732
C02344=1226.076,17.560,-42.432,-179.319,5.383,148.732
C02345=1226.070,17.809,-42.448,-179.316,5.383,148.731
C02346=1226.066,18.059,-42.462,-179.314,5.383,148.730
C02347=1226.061,18.309,-42.478,-179.311,5.384,148.730
C02348=1226.056,18.558,-42.493,-179.309,5.384,148.729
C02349=1226.050,18.807,-42.509,-179.306,5.385,148.728
C02350=1226.046,19.056,-42.524,-179.303,5.385,148.728
C02351=1226.040,19.306,-42.538,-179.301,5.385,148.727
C02352=1226.035,19.555,-42.553,-179.298,5.385,148.726
C02353=1226.031,19.806,-42.569,-179.296,5.386,148.726
C02354=1226.026,20.055,-42.584,-179.293,5.387,148.725
C02355=1226.021,20.304,-42.600,-179.291,5.387,148.724
C02356=1226.016,20.554,-42.614,-179.288,5.388,148.724
C02357=1226.010,20.803,-42.630,-179.286,5.387,148.723
C02358=1226.006,21.052,-42.645,-179.283,5.388,148.722
C02359=1226.001,21.302,-42.661,-179.281,5.388,148.722
C02360=1225.996,21.551,-42.676,-179.278,5.389,148.721
C02361=1225.991,21.801,-42.691,-179.276,5.390,148.720
C02362=1225.986,22.051,-42.706,-179.274,5.390,148.720
C02363=1225.981,22.300,-42.721,-179.271,5.390,148.719
C02364=1225.976,22.550,-42.737,-179.268,5.391,148.718
C02365=1225.971,22.799,-42.752,-179.266,5.391,148.718
C02366=1225.966,23.049,-42.768,-179.263,5.392,148.717
C02367=1225.961,23.298,-42.783,-179.260,5.392,148.716
C02368=1225.956,23.547,-42.798,-179.258,5.392,148.716
C02369=1225.951,23.797,-42.814,-179.256,5.393,148.715
C02370=1225.946,24.046,-42.829,-179.253,5.393,148.714
C02371=1225.941,24.296,-42.845,-179.250,5.394,148.714
C02372=1225.936,24.545,-42.860,-179.248,5.394,148.713
C02373=1225.931,24.795,-42.875,-179.245,5.395,148.712
C02374=1225.926,25.045,-42.891,-179.243,5.395,148.712
C02375=1225.921,25.294,-42.906,-179.240,5.395,148.711
C02376=1225.916,25.543,-42.921,-179.238,5.396,148.710
C02377=1225.910,25.793,-42.937,-179.235,5.396,148.709
C02378=1225.906,26.043,-42.952,-179.233,5.397,148.709
C02379=1225.901,26.292,-42.968,-179.230,5.398,148.708
C02380=1225.895,26.541,-42.983,-179.228,5.397,148.708
C02381=1225.891,26.790,-42.998,-179.226,5.398,148.707
C02382=1225.886,27.041,-43.014,-179.223,5.398,148.706
C02383=1225.881,27.290,-43.030,-179.220,5.399,148.706
C02384=1225.876,27.538,-43.046,-179.218,5.400,148.705
C02385=1225.872,27.789,-43.062,-179.215,5.400,148.704
C02386=1225.866,28.038,-43.077,-179.213,5.400,148.704
C02387=1225.861,28.287,-43.092,-179.210,5.400,148.703
C02388=1225.856,28.536,-43.108,-179.208,5.401,148.702
C02389=1225.851,28.787,-43.124,-179.205,5.401,148.702
C02390=1225.846,29.036,-43.139,-179.202,5.402,148.701
C02391=1225.841,29.304,-43.156,-179.200,5.403,148.700
C02392=1225.836,29.573,-43.173,-179.197,5.403,148.700
C02393=1225.830,29.842,-43.189,-179.194,5.404,148.699
C02394=1225.825,30.111,-43.206,-179.192,5.404,148.698
C02395=1225.820,30.360,-43.221,-179.189,5.405,148.697
C02396=1225.815,30.609,-43.238,-179.187,5.405,148.697
C02397=1225.810,30.859,-43.254,-179.184,5.405,148.696
C02398=1225.805,31.108,-43.269,-179.182,5.406,148.695
C02399=1225.800,31.357,-43.284,-179.179,5.406,148.695
C02400=1225.795,31.607,-43.300,-179.177,5.407,148.694
C02401=1225.790,31.857,-43.316,-179.174,5.407,148.693
C02402=1225.785,32.106,-43.332,-179.171,5.408,148.693
C02403=1225.780,32.356,-43.348,-179.169,5.408,148.692
C02404=1225.775,32.605,-43.363,-179.167,5.408,148.691
C02405=1225.770,32.854,-43.379,-179.164,5.409,148.691
C02406=1225.765,33.104,-43.395,-179.162,5.409,148.690
C02407=1225.760,33.353,-43.411,-179.159,5.410,148.690
C02408=1225.755,33.602,-43.426,-179.156,5.411,148.689
C02409=1225.751,33.852,-43.442,-179.154,5.411,148.688
C02410=1225.745,34.102,-43.457,-179.151,5.412,148.688
C02411=1225.740,34.350,-43.474,-179.149,5.412,148.687
C02412=1225.736,34.601,-43.490,-179.146,5.412,148.686
C02413=1225.730,34.850,-43.505,-179.144,5.413,148.686
C02414=1225.726,35.099,-43.522,-179.141,5.413,148.685
C02415=1225.720,35.349,-43.537,-179.139,5.414,148.684
C02416=1225.716,35.598,-43.552,-179.136,5.415,148.684
C02417=1225.711,35.848,-43.568,-179.134,5.415,148.683
C02418=1225.706,36.097,-43.585,-179.131,5.416,148.682
C02419=1225.701,36.347,-43.601,-179.128,5.416,148.682
C02420=1225.696,36.596,-43.616,-179.126,5.416,148.681
C02421=1225.691,36.845,-43.633,-179.124,5.416,148.680
C02422=1225.686,37.095,-43.649,-179.121,5.417,148.680
C02423=1225.681,37.344,-43.665,-179.118,5.418,148.679
C02424=1225.676,37.594,-43.681,-179.116,5.418,148.678
C02425=1225.670,37.844,-43.696,-179.113,5.419,148.678
C02426=1225.665,38.092,-43.713,-179.111,5.419,148.677
C02427=1225.661,38.342,-43.728,-179.108,5.420,148.677
C02428=1225.656,38.592,-43.744,-179.106,5.421,148.676
C02429=1225.651,38.841,-43.760,-179.104,5.420,148.675
C02430=1225.646,39.090,-43.776,-179.101,5.421,148.674
C02431=1225.642,39.340,-43.793,-179.098,5.422,148.674
C02432=1225.636,39.589,-43.808,-179.096,5.422,148.673
C02433=1225.631,39.838,-43.824,-179.093,5.423,148.672
C02434=1225.626,40.088,-43.840,-179.090,5.423,148.672
C02435=1225.621,40.337,-43.857,-179.088,5.424,148.671
C02436=1225.616,40.587,-43.873,-179.085,5.424,148.670
C02437=1225.611,40.836,-43.888,-179.083,5.425,148.670
C02438=1225.607,41.086,-43.905,-179.080,5.426,148.669
C02439=1225.601,41.335,-43.921,-179.078,5.426,148.669
C02440=1225.597,41.585,-43.937,-179.076,5.426,148.668
C02441=1225.591,41.834,-43.953,-179.073,5.427,148.667
C02442=1225.587,42.084,-43.969,-179.070,5.427,148.667
C02443=1225.582,42.332,-43.986,-179.068,5.428,148.666
C02444=1225.577,42.583,-44.002,-179.065,5.428,148.665
C02445=1225.572,42.831,-44.018,-179.062,5.429,148.665
C02446=1225.567,43.081,-44.034,-179.060,5.430,148.664
C02447=1225.562,43.330,-44.050,-179.058,5.430,148.664
C02448=1225.557,43.580,-44.066,-179.055,5.431,148.663
C02449=1225.551,43.829,-44.083,-179.052,5.432,148.662
C02450=1225.547,44.080,-44.099,-179.050,5.432,148.661
C02451=1225.542,44.328,-44.115,-179.048,5.432,148.661
C02452=1225.537,44.578,-44.132,-179.045,5.432,148.660
C02453=1225.532,44.827,-44.148,-179.042,5.433,148.659
C02454=1225.527,45.077,-44.164,-179.040,5.434,148.659
C02455=1225.522,45.325,-44.181,-179.038,5.434,148.658
C02456=1225.517,45.576,-44.197,-179.035,5.435,148.658
C02457=1225.512,45.824,-44.213,-179.032,5.436,148.657
C02458=1225.508,46.074,-44.229,-179.030,5.436,148.656
C02459=1225.503,46.324,-44.245,-179.027,5.437,148.656
C02460=1225.497,46.573,-44.262,-179.024,5.437,148.655
C02461=1225.492,46.823,-44.278,-179.022,5.438,148.654
C02462=1225.487,47.072,-44.295,-179.019,5.438,148.654
C02463=1225.483,47.321,-44.311,-179.017,5.439,148.653
C02464=1225.478,47.570,-44.328,-179.015,5.439,148.653
C02465=1225.473,47.820,-44.344,-179.012,5.440,148.652
C02466=1225.469,48.070,-44.360,-179.010,5.440,148.651
C02467=1225.463,48.319,-44.377,-179.007,5.441,148.651
C02468=1225.458,48.569,-44.393,-179.004,5.441,148.650
C02469=1225.453,48.818,-44.409,-179.002,5.442,148.649
C02470=1225.448,49.067,-44.426,-178.999,5.442,148.649
C02471=1225.444,49.317,-44.443,-178.997,5.443,148.648
C02472=1225.439,49.566,-44.458,-178.994,5.444,148.647
C02473=1225.433,49.816,-44.476,-178.992,5.444,148.647
C02474=1225.428,50.065,-44.492,-178.989,5.445,148.646
C02475=1225.424,50.314,-44.509,-178.986,5.446,148.645
C02476=1225.419,50.564,-44.525,-178.984,5.446,148.645
C02477=1225.413,50.813,-44.541,-178.981,5.447,148.644
C02478=1225.409,51.063,-44.558,-178.979,5.448,148.644
C02479=1225.404,51.312,-44.574,-178.976,5.448,148.643
C02480=1225.399,51.561,-44.591,-178.974,5.449,148.642
C02481=1225.395,51.811,-44.608,-178.972,5.449,148.642
C02482=1225.389,52.060,-44.625,-178.969,5.449,148.641
C02483=1225.384,52.310,-44.641,-178.966,5.450,148.640
C02484=1225.380,52.559,-44.657,-178.964,5.450,148.640
C02485=1225.374,52.808,-44.674,-178.961,5.451,148.639
C02486=1225.369,53.058,-44.691,-178.959,5.452,148.638
C02487=1225.365,53.307,-44.707,-178.956,5.452,148.638
C02488=1225.360,53.556,-44.724,-178.954,5.453,148.637
C02489=1225.354,53.806,-44.741,-178.951,5.453,148.636
C02490=1225.350,54.055,-44.758,-178.948,5.454,148.636
C02491=1225.345,54.304,-44.774,-178.946,5.455,148.635
C02492=1225.340,54.554,-44.791,-178.944,5.455,148.635
C02493=1225.335,54.804,-44.808,-178.941,5.456,148.634
C02494=1225.330,55.052,-44.824,-178.938,5.457,148.633
C02495=1225.324,55.322,-44.842,-178.936,5.457,148.633
C02496=1225.319,55.590,-44.860,-178.933,5.458,148.632
C02497=1225.315,55.858,-44.878,-178.931,5.458,148.631
C02498=1225.309,56.126,-44.896,-178.928,5.459,148.631
C02499=1225.304,56.376,-44.913,-178.925,5.459,148.630
C02500=1225.300,56.625,-44.930,-178.923,5.460,148.629
C02501=1225.294,56.874,-44.947,-178.920,5.461,148.629
C02502=1225.289,57.124,-44.963,-178.917,5.461,148.628
C02503=1225.284,57.374,-44.981,-178.915,5.462,148.627
C02504=1225.280,57.623,-44.997,-178.913,5.463,148.627
C02505=1225.274,57.872,-45.014,-178.910,5.463,148.626
C02506=1225.269,58.122,-45.031,-178.907,5.464,148.626
C02507=1225.265,58.371,-45.047,-178.905,5.464,148.625
C02508=1225.260,58.621,-45.065,-178.902,5.465,148.624
C02509=1225.254,58.870,-45.081,-178.899,5.466,148.624
C02510=1225.250,59.119,-45.098,-178.897,5.466,148.623
C02511=1225.245,59.369,-45.115,-178.895,5.467,148.622
C02512=1225.241,59.618,-45.132,-178.892,5.468,148.622
C02513=1225.235,59.867,-45.149,-178.889,5.468,148.621
C02514=1225.230,60.117,-45.166,-178.887,5.469,148.620
C02515=1225.225,60.366,-45.183,-178.884,5.469,148.620
C02516=1225.221,60.616,-45.200,-178.882,5.470,148.619
C02517=1225.215,60.865,-45.217,-178.879,5.471,148.619
C02518=1225.210,61.114,-45.233,-178.877,5.471,148.618
C02519=1225.206,61.363,-45.251,-178.874,5.472,148.617
C02520=1225.201,61.613,-45.268,-178.871,5.473,148.617
C02521=1225.196,61.862,-45.284,-178.869,5.473,148.616
C02522=1225.191,62.112,-45.302,-178.867,5.474,148.616
C02523=1225.186,62.361,-45.318,-178.864,5.475,148.615
C02524=1225.181,62.611,-45.336,-178.861,5.475,148.614
C02525=1225.177,62.860,-45.353,-178.859,5.476,148.614
C02526=1225.171,63.109,-45.370,-178.856,5.476,148.613
C02527=1225.166,63.358,-45.387,-178.853,5.477,148.612
C02528=1225.161,63.608,-45.404,-178.851,5.478,148.612
C02529=1225.156,63.857,-45.422,-178.849,5.478,148.611
C02530=1225.152,64.107,-45.438,-178.846,5.479,148.611
C02531=1225.147,64.357,-45.456,-178.843,5.480,148.610
C02532=1225.142,64.605,-45.472,-178.841,5.480,148.609
C02533=1225.137,64.855,-45.490,-178.839,5.481,148.609
C02534=1225.132,65.104,-45.507,-178.836,5.482,148.608
C02535=1225.127,65.354,-45.524,-178.833,5.482,148.607
C02536=1225.123,65.603,-45.541,-178.831,5.483,148.607
C02537=1225.118,65.853,-45.559,-178.828,5.483,148.606
C02538=1225.112,66.102,-45.575,-178.826,5.484,148.606
C02539=1225.108,66.350,-45.593,-178.823,5.485,148.605
C02540=1225.102,66.600,-45.610,-178.821,5.486,148.604
C02541=1225.098,66.850,-45.627,-178.818,5.486,148.604
C02542=1225.093,67.099,-45.645,-178.816,5.487,148.603
C02543=1225.088,67.349,-45.662,-178.813,5.487,148.602
C02544=1225.083,67.598,-45.679,-178.811,5.488,148.602
C02545=1225.078,67.847,-45.697,-178.808,5.489,148.601
C02546=1225.073,68.096,-45.713,-178.805,5.490,148.601
C02547=1225.068,68.345,-45.731,-178.802,5.491,148.600
C02548=1225.063,68.595,-45.748,-178.800,5.491,148.599
C02549=1225.059,68.844,-45.766,-178.798,5.492,148.599
C02550=1225.054,69.094,-45.783,-178.795,5.493,148.598
C02551=1225.049,69.344,-45.800,-178.792,5.493,148.598
C02552=1225.044,69.592,-45.818,-178.790,5.494,148.597
C02553=1225.039,69.842,-45.835,-178.787,5.495,148.596
C02554=1225.034,70.091,-45.853,-178.785,5.496,148.596
C02555=1225.030,70.341,-45.869,-178.782,5.496,148.595
C02556=1225.025,70.590,-45.887,-178.780,5.497,148.594
C02557=1225.019,70.839,-45.904,-178.777,5.497,148.594
C02558=1225.015,71.088,-45.922,-178.775,5.498,148.593
C02559=1225.010,71.338,-45.939,-178.772,5.499,148.593
C02560=1225.005,71.587,-45.957,-178.770,5.499,148.592
C02561=1224.999,71.837,-45.974,-178.767,5.500,148.591
C02562=1224.995,72.086,-45.992,-178.764,5.501,148.591
C02563=1224.990,72.336,-46.009,-178.762,5.501,148.590
C02564=1224.985,72.585,-46.027,-178.760,5.502,148.590
C02565=1224.980,72.834,-46.044,-178.757,5.503,148.589
C02566=1224.976,73.083,-46.061,-178.754,5.503,148.588
C02567=1224.971,73.333,-46.079,-178.752,5.504,148.588
C02568=1224.966,73.582,-46.097,-178.750,5.505,148.587
C02569=1224.961,73.831,-46.115,-178.746,5.506,148.587
C02570=1224.956,74.081,-46.131,-178.744,5.507,148.586
C02571=1224.951,74.330,-46.149,-178.741,5.507,148.585
C02572=1224.946,74.579,-46.167,-178.739,5.508,148.585
C02573=1224.941,74.829,-46.185,-178.736,5.509,148.584
C02574=1224.936,75.078,-46.203,-178.734,5.509,148.584
C02575=1224.932,75.327,-46.220,-178.731,5.510,148.583
C02576=1224.927,75.577,-46.237,-178.729,5.511,148.582
C02577=1224.922,75.826,-46.255,-178.726,5.512,148.582
C02578=1224.917,76.075,-46.273,-178.724,5.512,148.581
C02579=1224.912,76.325,-46.290,-178.721,5.513,148.580
C02580=1224.908,76.574,-46.308,-178.718,5.513,148.580
C02581=1224.903,76.823,-46.326,-178.716,5.514,148.579
C02582=1224.898,77.073,-46.343,-178.714,5.515,148.579
C02583=1224.893,77.322,-46.361,-178.711,5.515,148.578
C02584=1224.888,77.571,-46.379,-178.708,5.517,148.577
C02585=1224.883,77.821,-46.396,-178.706,5.518,148.577
C02586=1224.878,78.070,-46.414,-178.703,5.518,148.576
C02587=1224.873,78.319,-46.432,-178.700,5.519,148.576
C02588=1224.869,78.568,-46.450,-178.698,5.520,148.575
C02589=1224.864,78.817,-46.468,-178.696,5.521,148.575
C02590=1224.858,79.067,-46.485,-178.693,5.521,148.574
C02591=1224.853,79.316,-46.503,-178.690,5.522,148.573
C02592=1224.849,79.566,-46.521,-178.688,5.522,148.573
C02593=1224.844,79.815,-46.539,-178.686,5.523,148.572
C02594=1224.839,80.065,-46.557,-178.683,5.524,148.572
C02595=1224.834,80.314,-46.574,-178.680,5.524,148.571
C02596=1224.829,80.564,-46.592,-178.677,5.526,148.570
C02597=1224.824,80.813,-46.610,-178.675,5.527,148.570
C02598=1224.819,81.062,-46.628,-178.672,5.527,148.569
C02599=1224.814,81.330,-46.648,-178.670,5.528,148.568
C02600=1224.809,81.599,-46.666,-178.667,5.529,148.568
C02601=1224.804,81.867,-46.686,-178.664,5.530,148.567
C02602=1224.799,82.136,-46.705,-178.661,5.531,148.567
C02603=1224.794,82.385,-46.723,-178.659,5.531,148.566
C02604=1224.789,82.634,-46.741,-178.657,5.532,148.565
C02605=1224.784,82.883,-46.759,-178.654,5.533,148.565
C02606=1224.779,83.132,-46.777,-178.651,5.533,148.564
C02607=1224.774,83.382,-46.794,-178.649,5.534,148.563
C02608=1224.769,83.631,-46.812,-178.647,5.535,148.563
C02609=1224.764,83.880,-46.830,-178.643,5.536,148.562
C02610=1224.760,84.130,-46.849,-178.641,5.537,148.562
C02611=1224.755,84.380,-46.867,-178.638,5.537,148.561
C02612=1224.750,84.629,-46.885,-178.636,5.538,148.561
C02613=1224.745,84.878,-46.903,-178.633,5.539,148.560
C02614=1224.740,85.127,-46.921,-178.631,5.540,148.559
C02615=1224.735,85.376,-46.939,-178.629,5.540,148.559
C02616=1224.730,85.625,-46.957,-178.626,5.541,148.558
C02617=1224.726,85.875,-46.975,-178.623,5.542,148.558
C02618=1224.721,86.124,-46.993,-178.620,5.543,148.557
C02619=1224.716,86.374,-47.011,-178.618,5.544,148.557
C02620=1224.711,86.623,-47.029,-178.616,5.545,148.556
C02621=1224.706,86.872,-47.047,-178.613,5.545,148.555
C02622=1224.701,87.122,-47.066,-178.610,5.546,148.555
C02623=1224.697,87.371,-47.085,-178.608,5.547,148.554
C02624=1224.692,87.620,-47.103,-178.606,5.547,148.554
C02625=1224.687,87.869,-47.121,-178.603,5.548,148.553
C02626=1224.682,88.118,-47.139,-178.600,5.550,148.552
C02627=1224.677,88.367,-47.156,-178.598,5.550,148.552
C02628=1224.673,88.617,-47.175,-178.595,5.551,148.551
C02629=1224.668,88.866,-47.193,-178.592,5.552,148.551
C02630=1224.663,89.116,-47.211,-178.590,5.552,148.550
C02631=1224.657,89.365,-47.229,-178.588,5.553,148.549
C02632=1224.653,89.614,-47.248,-178.585,5.554,148.549
C02633=1224.648,89.864,-47.266,-178.582,5.555,148.548
C02634=1224.643,90.113,-47.284,-178.580,5.556,148.548
C02635=1224.638,90.362,-47.302,-178.577,5.557,148.547
C02636=1224.634,90.611,-47.320,-178.575,5.558,148.547
C02637=1224.629,90.861,-47.339,-178.572,5.558,148.546
C02638=1224.624,91.110,-47.358,-178.570,5.559,148.545
C02639=1224.619,91.359,-47.376,-178.567,5.559,148.545
C02640=1224.614,91.608,-47.394,-178.564,5.561,148.544
C02641=1224.610,91.858,-47.412,-178.562,5.562,148.544
C02642=1224.604,92.107,-47.432,-178.559,5.562,148.543
C02643=1224.600,92.356,-47.450,-178.557,5.563,148.543
C02644=1224.595,92.605,-47.468,-178.554,5.564,148.542
C02645=1224.590,92.855,-47.486,-178.552,5.564,148.541
C02646=1224.585,93.104,-47.505,-178.549,5.566,148.541
C02647=1224.580,93.353,-47.523,-178.546,5.567,148.540
C02648=1224.576,93.603,-47.541,-178.544,5.567,148.540
C02649=1224.571,93.852,-47.560,-178.541,5.568,148.539
C02650=1224.565,94.101,-47.579,-178.539,5.569,148.538
C02651=1224.561,94.350,-47.597,-178.536,5.570,148.538
C02652=1224.556,94.600,-47.615,-178.534,5.570,148.537
C02653=1224.552,94.849,-47.634,-178.531,5.572,148.537
C02654=1224.546,95.098,-47.652,-178.528,5.573,148.536
C02655=1224.542,95.347,-47.671,-178.526,5.573,148.535
C02656=1224.537,95.597,-47.689,-178.524,5.574,148.535
C02657=1224.531,95.846,-47.708,-178.521,5.575,148.534
C02658=1224.527,96.095,-47.727,-178.518,5.576,148.534
C02659=1224.523,96.345,-47.745,-178.516,5.577,148.533
C02660=1224.517,96.594,-47.764,-178.513,5.578,148.533
C02661=1224.513,96.843,-47.783,-178.511,5.578,148.532
C02662=1224.508,97.093,-47.801,-178.508,5.579,148.532
C02663=1224.503,97.341,-47.820,-178.506,5.580,148.531
C02664=1224.498,97.591,-47.838,-178.503,5.581,148.530
C02665=1224.494,97.840,-47.857,-178.500,5.582,148.530
C02666=1224.488,98.089,-47.876,-178.498,5.583,148.529
C02667=1224.484,98.339,-47.894,-178.495,5.583,148.529
C02668=1224.479,98.588,-47.913,-178.493,5.584,148.528
C02669=1224.473,98.837,-47.931,-178.490,5.586,148.528
C02670=1224.469,99.086,-47.950,-178.487,5.586,148.527
C02671=1224.464,99.336,-47.969,-178.485,5.587,148.526
C02672=1224.460,99.585,-47.988,-178.483,5.588,148.526
C02673=1224.455,99.834,-48.006,-178.480,5.589,148.525
C02674=1224.450,100.083,-48.025,-178.478,5.590,148.525
C02675=1224.445,100.333,-48.043,-178.475,5.591,148.524
C02676=1224.440,100.582,-48.063,-178.472,5.592,148.523
C02677=1224.436,100.831,-48.082,-178.470,5.593,148.523
C02678=1224.430,101.081,-48.100,-178.467,5.593,148.522
C02679=1224.426,101.329,-48.119,-178.465,5.594,148.522
C02680=1224.421,101.579,-48.137,-178.462,5.596,148.521
C02681=1224.416,101.828,-48.157,-178.459,5.596,148.521
C02682=1224.412,102.077,-48.176,-178.457,5.597,148.520
C02683=1224.406,102.327,-48.194,-178.455,5.598,148.520
C02684=1224.402,102.575,-48.213,-178.451,5.599,148.519
C02685=1224.397,102.826,-48.232,-178.449,5.600,148.518
C02686=1224.392,103.074,-48.251,-178.447,5.601,148.518
C02687=1224.387,103.324,-48.270,-178.444,5.601,148.517
C02688=1224.382,103.573,-48.288,-178.442,5.602,148.517
C02689=1224.378,103.822,-48.308,-178.439,5.604,148.516
C02690=1224.373,104.071,-48.327,-178.436,5.604,148.516
C02691=1224.368,104.321,-48.346,-178.434,5.605,148.515
C02692=1224.363,104.570,-48.364,-178.431,5.606,148.515
C02693=1224.358,104.819,-48.384,-178.429,5.607,148.514
C02694=1224.354,105.068,-48.402,-178.426,5.608,148.514
C02695=1224.348,105.317,-48.421,-178.424,5.609,148.513
C02696=1224.344,105.567,-48.441,-178.421,5.610,148.512
C02697=1224.339,105.815,-48.460,-178.419,5.611,148.512
C02698=1224.334,106.066,-48.479,-178.416,5.612,148.511
C02699=1224.329,106.314,-48.497,-178.413,5.613,148.511
C02700=1224.325,106.564,-48.517,-178.411,5.614,148.510
C02701=1224.320,106.812,-48.536,-178.408,5.614,148.509
C02702=1224.315,107.062,-48.555,-178.406,5.616,148.509
C02703=1224.310,107.330,-48.575,-178.403,5.617,148.508
C02704=1224.305,107.599,-48.596,-178.400,5.617,148.508
C02705=1224.300,107.867,-48.616,-178.397,5.619,148.507
C02706=1224.295,108.136,-48.637,-178.395,5.619,148.507
C02707=1224.289,108.385,-48.656,-178.392,5.620,148.506
C02708=1224.285,108.634,-48.676,-178.389,5.622,148.505
C02709=1224.280,108.883,-48.694,-178.387,5.623,148.505
C02710=1224.275,109.133,-48.713,-178.384,5.623,148.504
C02711=1224.270,109.382,-48.732,-178.382,5.624,148.504
C02712=1224.266,109.631,-48.752,-178.379,5.626,148.503
C02713=1224.261,109.881,-48.771,-178.377,5.626,148.503
C02714=1224.256,110.129,-48.790,-178.374,5.627,148.502
C02715=1224.251,110.379,-48.810,-178.372,5.628,148.502
C02716=1224.246,110.628,-48.829,-178.369,5.629,148.501
C02717=1224.242,110.877,-48.848,-178.367,5.630,148.501
C02718=1224.237,111.126,-48.867,-178.364,5.631,148.500
C02719=1224.232,111.376,-48.887,-178.361,5.631,148.499
C02720=1224.227,111.625,-48.907,-178.359,5.633,148.499
C02721=1224.222,111.874,-48.925,-178.356,5.634,148.498
C02722=1224.218,112.124,-48.944,-178.354,5.635,148.498
C02723=1224.212,112.373,-48.964,-178.351,5.635,148.497
C02724=1224.208,112.622,-48.983,-178.348,5.637,148.497
C02725=1224.203,112.871,-49.002,-178.346,5.638,148.496
C02726=1224.198,113.120,-49.022,-178.343,5.638,148.496
C02727=1224.193,113.370,-49.041,-178.341,5.640,148.495
C02728=1224.189,113.619,-49.060,-178.338,5.641,148.495
C02729=1224.184,113.868,-49.080,-178.336,5.642,148.494
C02730=1224.179,114.117,-49.099,-178.333,5.642,148.493
C02731=1224.174,114.366,-49.119,-178.330,5.644,148.493
C02732=1224.170,114.615,-49.139,-178.328,5.645,148.492
C02733=1224.165,114.864,-49.158,-178.325,5.645,148.492
C02734=1224.160,115.114,-49.177,-178.323,5.646,148.491
C02735=1224.155,115.363,-49.197,-178.320,5.648,148.491
C02736=1224.150,115.612,-49.216,-178.318,5.648,148.490
C02737=1224.145,115.862,-49.236,-178.315,5.649,148.490
C02738=1224.141,116.110,-49.255,-178.312,5.651,148.489
C02739=1224.136,116.360,-49.274,-178.310,5.652,148.489
C02740=1224.131,116.609,-49.294,-178.308,5.652,148.488
C02741=1224.126,116.858,-49.314,-178.305,5.653,148.488
C02742=1224.121,117.107,-49.334,-178.302,5.655,148.487
C02743=1224.117,117.357,-49.353,-178.300,5.655,148.486
C02744=1224.112,117.605,-49.372,-178.298,5.656,148.486
C02745=1224.107,117.855,-49.392,-178.294,5.658,148.485
C02746=1224.103,118.104,-49.411,-178.292,5.659,148.485
C02747=1224.098,118.353,-49.431,-178.290,5.659,148.484
C02748=1224.093,118.602,-49.451,-178.287,5.661,148.484
C02749=1224.088,118.852,-49.471,-178.284,5.662,148.483
C02750=1224.083,119.101,-49.490,-178.282,5.662,148.483
C02751=1224.078,119.350,-49.510,-178.280,5.663,148.482
C02752=1224.074,119.599,-49.530,-178.276,5.665,148.482
C02753=1224.070,119.848,-49.549,-178.274,5.666,148.481
C02754=1224.064,120.097,-49.568,-178.272,5.666,148.481
C02755=1224.059,120.347,-49.588,-178.269,5.668,148.480
C02756=1224.055,120.596,-49.608,-178.266,5.669,148.480
C02757=1224.050,120.845,-49.628,-178.264,5.670,148.479
C02758=1224.045,121.094,-49.647,-178.261,5.671,148.478
C02759=1224.041,121.343,-49.668,-178.258,5.672,148.478
C02760=1224.036,121.593,-49.687,-178.256,5.673,148.477
C02761=1224.030,121.842,-49.707,-178.253,5.674,148.477
C02762=1224.026,122.091,-49.727,-178.251,5.675,148.476
C02763=1224.021,122.340,-49.747,-178.248,5.676,148.476
C02764=1224.017,122.590,-49.766,-178.246,5.677,148.475
C02765=1224.011,122.838,-49.786,-178.243,5.678,148.475
C02766=1224.007,123.088,-49.806,-178.241,5.679,148.474
C02767=1224.002,123.337,-49.826,-178.238,5.680,148.474
C02768=1223.998,123.586,-49.846,-178.236,5.682,148.473
C02769=1223.992,123.835,-49.865,-178.233,5.682,148.473
C02770=1223.988,124.084,-49.886,-178.231,5.683,148.472
C02771=1223.983,124.333,-49.905,-178.228,5.685,148.472
C02772=1223.978,124.583,-49.925,-178.225,5.685,148.471
C02773=1223.974,124.832,-49.945,-178.223,5.686,148.471
C02774=1223.969,125.081,-49.965,-178.220,5.688,148.470
C02775=1223.964,125.330,-49.985,-178.218,5.689,148.470
C02776=1223.959,125.579,-50.005,-178.215,5.689,148.469
C02777=1223.955,125.828,-50.025,-178.213,5.691,148.469
C02778=1223.950,126.078,-50.045,-178.210,5.692,148.468
C02779=1223.945,126.326,-50.065,-178.208,5.693,148.467
C02780=1223.940,126.576,-50.085,-178.205,5.694,148.467
C02781=1223.935,126.825,-50.105,-178.203,5.695,148.466
C02782=1223.930,127.074,-50.125,-178.199,5.697,148.466
C02783=1223.926,127.323,-50.145,-178.197,5.698,148.465
C02784=1223.921,127.572,-50.165,-178.195,5.698,148.465
C02785=1223.916,127.821,-50.185,-178.192,5.700,148.464
C02786=1223.912,128.070,-50.205,-178.189,5.701,148.464
C02787=1223.907,128.320,-50.225,-178.187,5.702,148.463
C02788=1223.903,128.569,-50.245,-178.184,5.703,148.463
C02789=1223.897,128.819,-50.266,-178.182,5.704,148.462
C02790=1223.893,129.068,-50.286,-178.179,5.705,148.462
C02791=1223.887,129.316,-50.305,-178.177,5.707,148.461
C02792=1223.883,129.565,-50.326,-178.174,5.707,148.461
C02793=1223.878,129.814,-50.346,-178.172,5.708,148.460
C02794=1223.874,130.064,-50.366,-178.169,5.710,148.460
C02795=1223.869,130.313,-50.387,-178.167,5.711,148.459
C02796=1223.864,130.562,-50.407,-178.164,5.712,148.459
C02797=1223.859,130.812,-50.427,-178.161,5.713,148.458
C02798=1223.855,131.061,-50.447,-178.159,5.714,148.458
C02799=1223.850,131.309,-50.467,-178.156,5.715,148.457
C02800=1223.844,131.559,-50.487,-178.154,5.716,148.457
C02801=1223.840,131.808,-50.508,-178.151,5.717,148.456
C02802=1223.836,132.057,-50.528,-178.148,5.719,148.456
C02803=1223.831,132.306,-50.548,-178.146,5.720,148.455
C02804=1223.826,132.555,-50.569,-178.143,5.721,148.455
C02805=1223.821,132.804,-50.589,-178.141,5.722,148.454
C02806=1223.817,133.053,-50.609,-178.138,5.723,148.454
C02807=1223.811,133.322,-50.631,-178.135,5.724,148.453
C02808=1223.807,133.590,-50.653,-178.133,5.725,148.453
C02809=1223.801,133.859,-50.675,-178.130,5.726,148.452
C02810=1223.796,134.128,-50.697,-178.127,5.728,148.451
C02811=1223.792,134.377,-50.718,-178.125,5.729,148.451
C02812=1223.787,134.627,-50.737,-178.122,5.730,148.450
C02813=1223.781,134.875,-50.758,-178.119,5.731,148.450
C02814=1223.777,135.124,-50.778,-178.117,5.732,148.449
C02815=1223.772,135.373,-50.799,-178.114,5.734,148.449
C02816=1223.767,135.623,-50.820,-178.112,5.735,148.448
C02817=1223.763,135.872,-50.840,-178.109,5.735,148.448
C02818=1223.758,136.120,-50.860,-178.107,5.737,148.447
C02819=1223.753,136.370,-50.881,-178.104,5.738,148.447
C02820=1223.748,136.619,-50.901,-178.101,5.740,148.446
C02821=1223.744,136.868,-50.921,-178.099,5.740,148.446
C02822=1223.739,137.118,-50.942,-178.097,5.741,148.445
C02823=1223.734,137.366,-50.963,-178.094,5.743,148.445
C02824=1223.730,137.615,-50.983,-178.091,5.744,148.444
C02825=1223.725,137.865,-51.004,-178.088,5.745,148.444
C02826=1223.720,138.114,-51.024,-178.086,5.746,148.443
C02827=1223.715,138.363,-51.045,-178.084,5.747,148.443
C02828=1223.711,138.612,-51.066,-178.081,5.749,148.442
C02829=1223.706,138.861,-51.086,-178.079,5.750,148.442
C02830=1223.701,139.110,-51.107,-178.076,5.751,148.441
C02831=1223.697,139.359,-51.127,-178.073,5.752,148.441
C02832=1223.691,139.608,-51.148,-178.070,5.753,148.440
C02833=1223.687,139.857,-51.169,-178.068,5.754,148.440
C02834=1223.682,140.106,-51.190,-178.066,5.755,148.439
C02835=1223.677,140.355,-51.210,-178.063,5.757,148.439
C02836=1223.673,140.605,-51.231,-178.060,5.758,148.438
C02837=1223.668,140.854,-51.252,-178.058,5.759,148.438
C02838=1223.664,141.103,-51.272,-178.055,5.760,148.437
C02839=1223.659,141.353,-51.293,-178.052,5.762,148.437
C02840=1223.654,141.601,-51.314,-178.050,5.763,148.437
C02841=1223.649,141.851,-51.335,-178.048,5.763,148.436
C02842=1223.645,142.100,-51.355,-178.045,5.765,148.436
C02843=1223.639,142.349,-51.376,-178.042,5.766,148.435
C02844=1223.635,142.598,-51.396,-178.040,5.768,148.435
C02845=1223.630,142.847,-51.418,-178.037,5.768,148.434
C02846=1223.626,143.095,-51.438,-178.034,5.770,148.434
C02847=1223.621,143.345,-51.459,-178.032,5.771,148.433
C02848=1223.616,143.594,-51.480,-178.029,5.773,148.433
C02849=1223.612,143.844,-51.501,-178.027,5.774,148.432
C02850=1223.607,144.093,-51.521,-178.024,5.774,148.431
C02851=1223.602,144.341,-51.543,-178.022,5.776,148.431
C02852=1223.597,144.591,-51.564,-178.019,5.777,148.430
C02853=1223.593,144.839,-51.584,-178.017,5.778,148.430
C02854=1223.587,145.089,-51.605,-178.014,5.779,148.430
C02855=1223.583,145.338,-51.626,-178.011,5.781,148.429
C02856=1223.578,145.586,-51.647,-178.009,5.782,148.429
C02857=1223.574,145.836,-51.668,-178.006,5.783,148.428
C02858=1223.569,146.085,-51.689,-178.004,5.784,148.428
C02859=1223.564,146.334,-51.710,-178.001,5.786,148.427
C02860=1223.560,146.583,-51.731,-177.999,5.787,148.427
C02861=1223.555,146.832,-51.752,-177.997,5.788,148.426
C02862=1223.550,147.081,-51.773,-177.993,5.789,148.426
C02863=1223.545,147.330,-51.794,-177.991,5.790,148.425
C02864=1223.541,147.580,-51.816,-177.989,5.792,148.425
C02865=1223.536,147.829,-51.836,-177.986,5.793,148.424
C02866=1223.531,148.078,-51.857,-177.983,5.794,148.424
C02867=1223.526,148.326,-51.879,-177.981,5.795,148.423
C02868=1223.522,148.575,-51.899,-177.978,5.797,148.423
C02869=1223.517,148.824,-51.921,-177.976,5.798,148.423
C02870=1223.512,149.074,-51.942,-177.973,5.799,148.422
C02871=1223.508,149.323,-51.962,-177.971,5.800,148.422
C02872=1223.503,149.572,-51.984,-177.968,5.802,148.421
C02873=1223.498,149.821,-52.005,-177.965,5.803,148.421
C02874=1223.493,150.070,-52.025,-177.963,5.805,148.420
C02875=1223.489,150.319,-52.047,-177.960,5.805,148.420
C02876=1223.484,150.568,-52.068,-177.958,5.807,148.419
C02877=1223.479,150.817,-52.090,-177.955,5.808,148.419
C02878=1223.475,151.066,-52.110,-177.952,5.810,148.418
C02879=1223.470,151.315,-52.132,-177.950,5.811,148.418
C02880=1223.465,151.565,-52.153,-177.947,5.812,148.417
C02881=1223.460,151.813,-52.175,-177.945,5.813,148.417
C02882=1223.456,152.062,-52.195,-177.942,5.815,148.416
C02883=1223.451,152.311,-52.217,-177.940,5.815,148.416
C02884=1223.447,152.561,-52.238,-177.937,5.817,148.415
C02885=1223.442,152.809,-52.260,-177.934,5.818,148.415
C02886=1223.437,153.058,-52.281,-177.932,5.820,148.414
C02887=1223.432,153.307,-52.302,-177.930,5.821,148.414
C02888=1223.428,153.557,-52.324,-177.926,5.822,148.413
C02889=1223.423,153.806,-52.345,-177.924,5.823,148.413
C02890=1223.418,154.055,-52.366,-177.922,5.825,148.413
C02891=1223.413,154.304,-52.388,-177.919,5.826,148.412
C02892=1223.409,154.553,-52.409,-177.916,5.827,148.412
C02893=1223.404,154.802,-52.430,-177.914,5.828,148.411
C02894=1223.399,155.050,-52.452,-177.911,5.830,148.411
C02895=1223.395,155.300,-52.473,-177.909,5.831,148.410
C02896=1223.390,155.549,-52.495,-177.906,5.832,148.410
C02897=1223.385,155.798,-52.517,-177.904,5.833,148.409
C02898=1223.381,156.047,-52.537,-177.901,5.835,148.409
C02899=1223.376,156.296,-52.559,-177.899,5.836,148.408
C02900=1223.371,156.545,-52.580,-177.896,5.838,148.408
C02901=1223.367,156.795,-52.602,-177.894,5.839,148.408
C02902=1223.362,157.043,-52.624,-177.891,5.840,148.407
C02903=1223.357,157.292,-52.645,-177.889,5.841,148.407
C02904=1223.352,157.541,-52.666,-177.886,5.843,148.406
C02905=1223.348,157.790,-52.688,-177.883,5.844,148.406
C02906=1223.343,158.039,-52.710,-177.881,5.845,148.405
C02907=1223.338,158.289,-52.732,-177.878,5.847,148.405
C02908=1223.334,158.537,-52.753,-177.875,5.848,148.404
C02909=1223.329,158.786,-52.774,-177.873,5.850,148.404
C02910=1223.325,159.035,-52.796,-177.871,5.851,148.403
C02911=1223.319,159.305,-52.820,-177.867,5.852,148.403
C02912=1223.314,159.574,-52.843,-177.865,5.854,148.402
C02913=1223.310,159.843,-52.867,-177.862,5.855,148.402
C02914=1223.304,160.112,-52.890,-177.859,5.856,148.401
C02915=1223.299,160.361,-52.912,-177.856,5.858,148.401
C02916=1223.295,160.610,-52.934,-177.854,5.859,148.401
C02917=1223.290,160.859,-52.955,-177.851,5.860,148.400
C02918=1223.285,161.108,-52.976,-177.849,5.861,148.400
C02919=1223.281,161.357,-52.998,-177.846,5.863,148.399
C02920=1223.276,161.606,-53.020,-177.844,5.865,148.399
C02921=1223.271,161.854,-53.042,-177.841,5.866,148.398
C02922=1223.267,162.104,-53.064,-177.838,5.868,148.398
C02923=1223.262,162.352,-53.085,-177.836,5.869,148.397
C02924=1223.257,162.602,-53.107,-177.833,5.870,148.397
C02925=1223.253,162.850,-53.129,-177.831,5.871,148.396
C02926=1223.248,163.100,-53.150,-177.828,5.873,148.396
C02927=1223.243,163.349,-53.172,-177.826,5.874,148.395
C02928=1223.238,163.598,-53.194,-177.823,5.875,148.395
C02929=1223.234,163.847,-53.216,-177.821,5.877,148.395
C02930=1223.229,164.096,-53.238,-177.818,5.878,148.394
C02931=1223.225,164.345,-53.260,-177.815,5.880,148.394
C02932=1223.220,164.594,-53.281,-177.813,5.881,148.393
C02933=1223.215,164.843,-53.304,-177.811,5.882,148.393
C02934=1223.210,165.092,-53.326,-177.807,5.884,148.392
C02935=1223.206,165.341,-53.348,-177.805,5.885,148.392
C02936=1223.201,165.590,-53.369,-177.803,5.887,148.392
C02937=1223.197,165.839,-53.391,-177.800,5.887,148.391
C02938=1223.192,166.088,-53.413,-177.797,5.889,148.391
C02939=1223.188,166.337,-53.435,-177.795,5.890,148.390
C02940=1223.183,166.586,-53.457,-177.792,5.892,148.390
C02941=1223.178,166.835,-53.480,-177.790,5.894,148.389
C02942=1223.173,167.083,-53.502,-177.787,5.895,148.389
C02943=1223.169,167.333,-53.524,-177.785,5.896,148.389
C02944=1223.164,167.581,-53.546,-177.782,5.897,148.388
C02945=1223.160,167.831,-53.568,-177.780,5.899,148.388
C02946=1223.155,168.079,-53.589,-177.777,5.901,148.387
C02947=1223.150,168.329,-53.612,-177.774,5.901,148.387
C02948=1223.145,168.578,-53.634,-177.772,5.903,148.386
C02949=1223.141,168.827,-53.656,-177.770,5.904,148.386
C02950=1223.136,169.075,-53.678,-177.767,5.906,148.386
C02951=1223.131,169.325,-53.701,-177.764,5.907,148.385
C02952=1223.126,169.573,-53.722,-177.762,5.908,148.385
C02953=1223.122,169.823,-53.744,-177.759,5.910,148.384
C02954=1223.117,170.071,-53.766,-177.757,5.911,148.384
C02955=1223.113,170.320,-53.789,-177.754,5.913,148.383
C02956=1223.108,170.569,-53.811,-177.751,5.915,148.383
C02957=1223.103,170.818,-53.833,-177.749,5.916,148.382
C02958=1223.098,171.067,-53.855,-177.746,5.917,148.382
C02959=1223.094,171.316,-53.878,-177.743,5.919,148.381
C02960=1223.090,171.565,-53.900,-177.741,5.920,148.381
C02961=1223.085,171.814,-53.922,-177.738,5.922,148.381
C02962=1223.080,172.063,-53.944,-177.736,5.922,148.380
C02963=1223.075,172.312,-53.967,-177.733,5.924,148.380
C02964=1223.071,172.561,-53.989,-177.731,5.926,148.379
C02965=1223.067,172.810,-54.011,-177.728,5.927,148.379
C02966=1223.061,173.059,-54.034,-177.725,5.929,148.378
C02967=1223.057,173.308,-54.056,-177.723,5.930,148.378
C02968=1223.052,173.557,-54.078,-177.721,5.931,148.378
C02969=1223.047,173.806,-54.101,-177.718,5.933,148.377
C02970=1223.043,174.055,-54.123,-177.715,5.934,148.377
C02971=1223.038,174.304,-54.145,-177.713,5.936,148.376
C02972=1223.034,174.553,-54.168,-177.710,5.938,148.376
C02973=1223.029,174.801,-54.190,-177.708,5.939,148.376
C02974=1223.024,175.050,-54.213,-177.705,5.940,148.375
C02975=1223.020,175.300,-54.235,-177.702,5.942,148.375
C02976=1223.015,175.548,-54.257,-177.700,5.943,148.374
C02977=1223.010,175.797,-54.280,-177.697,5.945,148.374
C02978=1223.006,176.047,-54.302,-177.695,5.947,148.374
C02979=1223.001,176.295,-54.325,-177.692,5.947,148.373
C02980=1222.996,176.544,-54.348,-177.689,5.949,148.373
C02981=1222.992,176.793,-54.370,-177.687,5.951,148.372
C02982=1222.987,177.042,-54.393,-177.685,5.952,148.372
C02983=1222.983,177.291,-54.415,-177.682,5.953,148.371
C02984=1222.978,177.540,-54.438,-177.679,5.955,148.371
C02985=1222.973,177.788,-54.460,-177.677,5.956,148.371
C02986=1222.968,178.038,-54.483,-177.674,5.958,148.370
C02987=1222.964,178.287,-54.506,-177.672,5.959,148.370
C02988=1222.959,178.536,-54.528,-177.669,5.961,148.369
C02989=1222.955,178.785,-54.551,-177.666,5.962,148.369
C02990=1222.950,179.034,-54.573,-177.664,5.963,148.368
C02991=1222.945,179.282,-54.596,-177.662,5.965,148.368
C02992=1222.940,179.531,-54.619,-177.658,5.967,148.368
C02993=1222.936,179.781,-54.641,-177.656,5.969,148.367
C02994=1222.931,180.030,-54.665,-177.654,5.970,148.367
C02995=1222.927,180.278,-54.686,-177.651,5.971,148.366
C02996=1222.922,180.527,-54.710,-177.648,5.973,148.366
C02997=1222.918,180.776,-54.732,-177.646,5.974,148.366
C02998=1222.912,181.025,-54.755,-177.643,5.976,148.365
C02999=1222.908,181.274,-54.777,-177.640,5.978,148.365
C03000=1222.904,181.523,-54.801,-177.638,5.979,148.364
C03001=1222.899,181.772,-54.823,-177.636,5.980,148.364
C03002=1222.894,182.020,-54.846,-177.633,5.982,148.363
C03003=1222.889,182.269,-54.869,-177.631,5.983,148.363
C03004=1222.885,182.518,-54.892,-177.628,5.985,148.363
C03005=1222.880,182.768,-54.915,-177.625,5.987,148.362
C03006=1222.876,183.017,-54.937,-177.623,5.988,148.362
C03007=1222.871,183.265,-54.960,-177.620,5.989,148.361
C03008=1222.866,183.515,-54.983,-177.617,5.991,148.361
C03009=1222.862,183.763,-55.006,-177.615,5.993,148.361
C03010=1222.857,184.012,-55.029,-177.613,5.994,148.360
C03011=1222.853,184.260,-55.052,-177.610,5.996,148.360
C03012=1222.848,184.509,-55.075,-177.607,5.997,148.360
C03013=1222.843,184.759,-55.098,-177.605,5.998,148.359
C03014=1222.839,185.008,-55.120,-177.602,6.000,148.359
C03015=1222.834,185.277,-55.145,-177.599,6.002,148.358
C03016=1222.829,185.547,-55.170,-177.596,6.003,148.358
C03017=1222.824,185.817,-55.195,-177.594,6.005,148.357
C03018=1222.819,186.086,-55.221,-177.591,6.007,148.357
C03019=1222.814,186.335,-55.243,-177.589,6.008,148.357
C03020=1222.810,186.584,-55.266,-177.586,6.009,148.356
C03021=1222.805,186.833,-55.289,-177.583,6.011,148.356
C03022=1222.800,187.082,-55.312,-177.580,6.013,148.355
C03023=1222.795,187.331,-55.336,-177.578,6.014,148.355
C03024=1222.791,187.579,-55.358,-177.576,6.016,148.355
C03025=1222.787,187.828,-55.382,-177.573,6.018,148.354
C03026=1222.782,188.077,-55.405,-177.570,6.019,148.354
C03027=1222.778,188.326,-55.428,-177.568,6.020,148.353
C03028=1222.773,188.574,-55.451,-177.565,6.022,148.353
C03029=1222.768,188.823,-55.474,-177.563,6.024,148.353
C03030=1222.763,189.072,-55.498,-177.560,6.025,148.352
C03031=1222.759,189.322,-55.521,-177.558,6.027,148.352
C03032=1222.755,189.570,-55.544,-177.555,6.029,148.352
C03033=1222.750,189.819,-55.567,-177.552,6.030,148.351
C03034=1222.745,190.068,-55.591,-177.550,6.031,148.351
C03035=1222.741,190.317,-55.614,-177.547,6.033,148.350
C03036=1222.736,190.566,-55.637,-177.545,6.035,148.350
C03037=1222.731,190.814,-55.660,-177.542,6.037,148.350
C03038=1222.727,191.063,-55.683,-177.540,6.038,148.349
C03039=1222.722,191.312,-55.706,-177.537,6.040,148.349
C03040=1222.717,191.561,-55.730,-177.534,6.041,148.348
C03041=1222.712,191.811,-55.753,-177.532,6.043,148.348
C03042=1222.708,192.060,-55.776,-177.529,6.044,148.348
C03043=1222.704,192.308,-55.799,-177.527,6.046,148.347
C03044=1222.699,192.557,-55.823,-177.524,6.048,148.347
C03045=1222.695,192.806,-55.847,-177.522,6.049,148.347
C03046=1222.690,193.055,-55.870,-177.519,6.050,148.346
C03047=1222.685,193.304,-55.893,-177.516,6.052,148.346
C03048=1222.681,193.553,-55.917,-177.514,6.054,148.345
C03049=1222.676,193.802,-55.940,-177.511,6.056,148.345
C03050=1222.672,194.050,-55.964,-177.509,6.057,148.345
C03051=1222.667,194.299,-55.987,-177.506,6.058,148.344
C03052=1222.662,194.548,-56.010,-177.504,6.060,148.344
C03053=1222.657,194.797,-56.034,-177.501,6.062,148.344
C03054=1222.653,195.045,-56.057,-177.498,6.064,148.343
C03055=1222.648,195.294,-56.081,-177.496,6.065,148.343
C03056=1222.644,195.543,-56.104,-177.493,6.067,148.342
C03057=1222.639,195.792,-56.127,-177.490,6.068,148.342
C03058=1222.634,196.041,-56.151,-177.488,6.070,148.342
C03059=1222.630,196.289,-56.175,-177.486,6.071,148.341
C03060=1222.625,196.538,-56.198,-177.483,6.073,148.341
C03061=1222.621,196.787,-56.222,-177.480,6.075,148.340
C03062=1222.616,197.036,-56.246,-177.478,6.077,148.340
C03063=1222.612,197.285,-56.269,-177.475,6.079,148.340
C03064=1222.607,197.534,-56.292,-177.473,6.080,148.339
C03065=1222.602,197.782,-56.316,-177.470,6.081,148.339
C03066=1222.598,198.032,-56.340,-177.467,6.083,148.338
C03067=1222.594,198.281,-56.363,-177.465,6.085,148.338
C03068=1222.589,198.529,-56.388,-177.462,6.087,148.338
C03069=1222.585,198.778,-56.411,-177.460,6.088,148.337
C03070=1222.580,199.027,-56.435,-177.457,6.090,148.337
C03071=1222.575,199.276,-56.459,-177.455,6.091,148.337
C03072=1222.570,199.525,-56.482,-177.452,6.093,148.336
C03073=1222.566,199.774,-56.506,-177.449,6.095,148.336
C03074=1222.561,200.023,-56.530,-177.447,6.096,148.336
C03075=1222.556,200.271,-56.554,-177.445,6.098,148.335
C03076=1222.552,200.520,-56.577,-177.442,6.100,148.335
C03077=1222.547,200.769,-56.601,-177.439,6.101,148.334
C03078=1222.543,201.018,-56.625,-177.436,6.103,148.334
C03079=1222.538,201.266,-56.649,-177.434,6.104,148.334
C03080=1222.534,201.515,-56.672,-177.432,6.106,148.333
C03081=1222.530,201.764,-56.696,-177.429,6.108,148.333
C03082=1222.524,202.013,-56.720,-177.426,6.110,148.333
C03083=1222.520,202.262,-56.745,-177.424,6.112,148.332
C03084=1222.515,202.511,-56.768,-177.421,6.113,148.332
C03085=1222.511,202.759,-56.792,-177.419,6.114,148.332
C03086=1222.506,203.008,-56.816,-177.416,6.116,148.331
C03087=1222.502,203.257,-56.839,-177.414,6.118,148.331
C03088=1222.497,203.506,-56.864,-177.411,6.120,148.331
C03089=1222.492,203.755,-56.887,-177.408,6.122,148.330
C03090=1222.488,204.004,-56.912,-177.406,6.124,148.330
C03091=1222.484,204.252,-56.936,-177.404,6.125,148.330
C03092=1222.479,204.501,-56.959,-177.401,6.126,148.329
C03093=1222.474,204.750,-56.984,-177.398,6.128,148.329
C03094=1222.469,204.999,-57.007,-177.395,6.130,148.328
C03095=1222.465,205.247,-57.031,-177.393,6.132,148.328
C03096=1222.461,205.496,-57.056,-177.390,6.134,148.328
C03097=1222.457,205.745,-57.080,-177.388,6.135,148.327
C03098=1222.451,205.994,-57.104,-177.385,6.136,148.327
C03099=1222.447,206.243,-57.128,-177.383,6.138,148.327
C03100=1222.442,206.491,-57.152,-177.380,6.140,148.326
C03101=1222.437,206.740,-57.176,-177.377,6.142,148.326
C03102=1222.433,206.989,-57.200,-177.375,6.144,148.326
C03103=1222.429,207.238,-57.224,-177.373,6.145,148.325
C03104=1222.424,207.486,-57.249,-177.370,6.147,148.325
C03105=1222.419,207.736,-57.273,-177.367,6.149,148.325
C03106=1222.415,207.984,-57.297,-177.365,6.150,148.324
C03107=1222.411,208.233,-57.321,-177.362,6.152,148.324
C03108=1222.406,208.482,-57.346,-177.359,6.154,148.324
C03109=1222.401,208.730,-57.370,-177.357,6.156,148.323
C03110=1222.397,208.979,-57.393,-177.354,6.158,148.323
C03111=1222.391,209.228,-57.418,-177.352,6.159,148.323
C03112=1222.388,209.477,-57.442,-177.349,6.161,148.322
C03113=1222.383,209.726,-57.466,-177.347,6.162,148.322
C03114=1222.378,209.974,-57.491,-177.344,6.164,148.322
C03115=1222.374,210.223,-57.515,-177.342,6.166,148.321
C03116=1222.369,210.472,-57.540,-177.339,6.168,148.321
C03117=1222.365,210.721,-57.564,-177.336,6.170,148.321
C03118=1222.360,210.970,-57.588,-177.334,6.171,148.320
C03119=1222.355,211.240,-57.614,-177.331,6.173,148.320
C03120=1222.350,211.511,-57.641,-177.328,6.175,148.319
C03121=1222.345,211.781,-57.668,-177.325,6.177,148.319
C03122=1222.340,212.052,-57.694,-177.323,6.179,148.319
C03123=1222.335,212.300,-57.718,-177.320,6.181,148.318
C03124=1222.332,212.549,-57.743,-177.317,6.183,148.318
C03125=1222.326,212.798,-57.767,-177.315,6.184,148.318
C03126=1222.322,213.046,-57.791,-177.312,6.186,148.317
C03127=1222.318,213.296,-57.816,-177.310,6.187,148.317
C03128=1222.313,213.544,-57.840,-177.307,6.189,148.317
C03129=1222.308,213.793,-57.865,-177.305,6.191,148.316
C03130=1222.304,214.041,-57.890,-177.302,6.193,148.316
C03131=1222.299,214.290,-57.915,-177.299,6.195,148.316
C03132=1222.295,214.538,-57.939,-177.297,6.197,148.315
C03133=1222.290,214.787,-57.964,-177.294,6.198,148.315
C03134=1222.286,215.036,-57.988,-177.292,6.200,148.315
C03135=1222.281,215.285,-58.013,-177.289,6.202,148.314
C03136=1222.277,215.533,-58.037,-177.286,6.204,148.314
C03137=1222.272,215.783,-58.062,-177.284,6.206,148.314
C03138=1222.268,216.031,-58.086,-177.282,6.207,148.313
C03139=1222.263,216.281,-58.111,-177.279,6.209,148.313
C03140=1222.259,216.528,-58.136,-177.276,6.211,148.313
C03141=1222.254,216.777,-58.160,-177.274,6.212,148.312
C03142=1222.249,217.027,-58.185,-177.271,6.214,148.312
C03143=1222.245,217.275,-58.210,-177.268,6.216,148.312
C03144=1222.240,217.524,-58.234,-177.266,6.218,148.311
C03145=1222.236,217.772,-58.259,-177.263,6.220,148.311
C03146=1222.231,218.021,-58.284,-177.261,6.222,148.311
C03147=1222.227,218.270,-58.309,-177.258,6.224,148.310
C03148=1222.222,218.519,-58.333,-177.255,6.225,148.310
C03149=1222.217,218.767,-58.358,-177.253,6.227,148.310
C03150=1222.214,219.016,-58.383,-177.251,6.228,148.309
C03151=1222.209,219.265,-58.408,-177.248,6.230,148.309
C03152=1222.204,219.514,-58.433,-177.245,6.232,148.309
C03153=1222.200,219.762,-58.457,-177.243,6.234,148.308
C03154=1222.195,220.011,-58.482,-177.240,6.236,148.308
C03155=1222.190,220.260,-58.507,-177.238,6.238,148.308
C03156=1222.186,220.508,-58.532,-177.235,6.240,148.307
C03157=1222.182,220.757,-58.557,-177.233,6.242,148.307
C03158=1222.176,221.006,-58.582,-177.230,6.243,148.307
C03159=1222.173,221.254,-58.607,-177.227,6.245,148.306
C03160=1222.168,221.503,-58.631,-177.225,6.247,148.306
C03161=1222.163,221.753,-58.657,-177.222,6.249,148.306
C03162=1222.159,222.000,-58.681,-177.220,6.251,148.306
C03163=1222.154,222.249,-58.706,-177.217,6.253,148.305
C03164=1222.150,222.498,-58.732,-177.214,6.255,148.305
C03165=1222.145,222.747,-58.756,-177.212,6.256,148.304
C03166=1222.141,222.996,-58.781,-177.210,6.257,148.304
C03167=1222.136,223.244,-58.806,-177.207,6.259,148.304
C03168=1222.132,223.493,-58.831,-177.204,6.261,148.304
C03169=1222.127,223.741,-58.857,-177.202,6.263,148.303
C03170=1222.123,223.991,-58.881,-177.200,6.265,148.303
C03171=1222.118,224.239,-58.906,-177.197,6.267,148.303
C03172=1222.114,224.488,-58.931,-177.194,6.269,148.302
C03173=1222.109,224.736,-58.957,-177.192,6.271,148.302
C03174=1222.104,224.986,-58.982,-177.189,6.273,148.302
C03175=1222.100,225.233,-59.007,-177.186,6.275,148.301
C03176=1222.096,225.483,-59.032,-177.184,6.276,148.301
C03177=1222.091,225.731,-59.057,-177.181,6.278,148.301
C03178=1222.087,225.980,-59.083,-177.179,6.280,148.300
C03179=1222.081,226.228,-59.108,-177.176,6.282,148.300
C03180=1222.077,226.477,-59.133,-177.173,6.284,148.300
C03181=1222.073,226.726,-59.158,-177.171,6.286,148.300
C03182=1222.069,226.974,-59.183,-177.169,6.288,148.299
C03183=1222.064,227.223,-59.209,-177.166,6.290,148.299
C03184=1222.059,227.472,-59.234,-177.163,6.292,148.299
C03185=1222.055,227.721,-59.259,-177.161,6.293,148.298
C03186=1222.050,227.970,-59.284,-177.159,6.295,148.298
C03187=1222.046,228.218,-59.310,-177.156,6.296,148.298
C03188=1222.041,228.466,-59.335,-177.153,6.298,148.297
C03189=1222.037,228.715,-59.360,-177.151,6.300,148.297
C03190=1222.033,228.964,-59.385,-177.149,6.302,148.297
C03191=1222.028,229.212,-59.411,-177.146,6.304,148.297
C03192=1222.024,229.461,-59.436,-177.143,6.306,148.296
C03193=1222.019,229.710,-59.461,-177.141,6.308,148.296
C03194=1222.014,229.959,-59.487,-177.138,6.310,148.296
C03195=1222.010,230.208,-59.513,-177.135,6.312,148.295
C03196=1222.005,230.456,-59.538,-177.133,6.313,148.295
C03197=1222.001,230.705,-59.563,-177.131,6.316,148.295
C03198=1221.996,230.953,-59.588,-177.128,6.318,148.295
C03199=1221.992,231.202,-59.614,-177.125,6.319,148.294
C03200=1221.988,231.451,-59.640,-177.123,6.321,148.294
C03201=1221.983,231.699,-59.665,-177.120,6.323,148.294
C03202=1221.978,231.948,-59.690,-177.118,6.325,148.293
C03203=1221.974,232.197,-59.716,-177.115,6.327,148.293
C03204=1221.969,232.445,-59.741,-177.113,6.329,148.293
C03205=1221.965,232.694,-59.767,-177.110,6.331,148.293
C03206=1221.961,232.943,-59.793,-177.108,6.333,148.292
C03207=1221.956,233.191,-59.818,-177.105,6.335,148.292
C03208=1221.952,233.440,-59.844,-177.102,6.336,148.292
C03209=1221.947,233.689,-59.870,-177.100,6.338,148.291
C03210=1221.943,233.937,-59.895,-177.098,6.341,148.291
C03211=1221.938,234.186,-59.920,-177.095,6.342,148.291
C03212=1221.934,234.435,-59.946,-177.092,6.344,148.291
C03213=1221.929,234.683,-59.971,-177.090,6.346,148.290
C03214=1221.924,234.932,-59.998,-177.087,6.348,148.290
C03215=1221.920,235.181,-60.023,-177.084,6.350,148.290
C03216=1221.915,235.429,-60.049,-177.082,6.352,148.290
C03217=1221.911,235.678,-60.075,-177.080,6.354,148.289
C03218=1221.907,235.927,-60.100,-177.077,6.356,148.289
C03219=1221.902,236.175,-60.126,-177.074,6.358,148.289
C03220=1221.898,236.424,-60.152,-177.072,6.360,148.288
C03221=1221.893,236.672,-60.177,-177.069,6.361,148.288
C03222=1221.888,236.922,-60.204,-177.067,6.364,148.288
C03223=1221.883,237.192,-60.232,-177.064,6.365,148.288
C03224=1221.879,237.464,-60.260,-177.062,6.367,148.287
C03225=1221.873,237.735,-60.288,-177.059,6.370,148.287
C03226=1221.869,238.006,-60.316,-177.056,6.372,148.287
C03227=1221.865,238.255,-60.342,-177.053,6.374,148.286
C03228=1221.860,238.503,-60.368,-177.051,6.376,148.286
C03229=1221.856,238.752,-60.393,-177.048,6.377,148.286
C03230=1221.851,239.001,-60.420,-177.046,6.380,148.286
C03231=1221.847,239.250,-60.445,-177.043,6.382,148.285
C03232=1221.843,239.498,-60.472,-177.041,6.383,148.285
C03233=1221.838,239.746,-60.497,-177.038,6.385,148.285
C03234=1221.833,239.995,-60.524,-177.035,6.387,148.284
C03235=1221.829,240.244,-60.549,-177.033,6.389,148.284
C03236=1221.824,240.493,-60.575,-177.031,6.391,148.284
C03237=1221.820,240.741,-60.601,-177.028,6.393,148.284
C03238=1221.815,240.990,-60.628,-177.026,6.395,148.283
C03239=1221.811,241.239,-60.653,-177.023,6.397,148.283
C03240=1221.806,241.487,-60.679,-177.021,6.399,148.283
C03241=1221.802,241.736,-60.706,-177.018,6.401,148.283
C03242=1221.797,241.984,-60.732,-177.016,6.403,148.282
C03243=1221.793,242.233,-60.757,-177.012,6.405,148.282
C03244=1221.789,242.482,-60.783,-177.010,6.408,148.282
C03245=1221.784,242.730,-60.810,-177.008,6.410,148.282
C03246=1221.780,242.979,-60.836,-177.005,6.411,148.281
C03247=1221.775,243.228,-60.862,-177.002,6.413,148.281
C03248=1221.770,243.475,-60.888,-177.000,6.415,148.281
C03249=1221.766,243.724,-60.914,-176.998,6.417,148.281
C03250=1221.762,243.973,-60.940,-176.995,6.419,148.280
C03251=1221.757,244.222,-60.967,-176.992,6.421,148.280
C03252=1221.753,244.470,-60.993,-176.990,6.423,148.280
C03253=1221.748,244.719,-61.020,-176.988,6.425,148.280
C03254=1221.744,244.968,-61.045,-176.985,6.427,148.279
C03255=1221.740,245.216,-61.071,-176.982,6.429,148.279
C03256=1221.734,245.464,-61.098,-176.980,6.431,148.279
C03257=1221.730,245.713,-61.124,-176.978,6.433,148.278
C03258=1221.726,245.962,-61.151,-176.975,6.435,148.278
C03259=1221.721,246.210,-61.176,-176.972,6.437,148.278
C03260=1221.717,246.459,-61.203,-176.970,6.439,148.278
C03261=1221.712,246.708,-61.229,-176.968,6.441,148.277
C03262=1221.709,246.956,-61.256,-176.965,6.443,148.277
C03263=1221.704,247.205,-61.282,-176.962,6.445,148.277
C03264=1221.700,247.453,-61.309,-176.960,6.448,148.277
C03265=1221.695,247.702,-61.335,-176.957,6.449,148.276
C03266=1221.690,247.950,-61.361,-176.954,6.451,148.276
C03267=1221.685,248.199,-61.387,-176.952,6.453,148.276
C03268=1221.681,248.447,-61.414,-176.950,6.455,148.276
C03269=1221.676,248.696,-61.440,-176.947,6.457,148.275
C03270=1221.672,248.944,-61.467,-176.945,6.459,148.275
C03271=1221.668,249.193,-61.494,-176.942,6.461,148.275
C03272=1221.664,249.442,-61.519,-176.940,6.463,148.275
C03273=1221.659,249.690,-61.546,-176.937,6.465,148.274
C03274=1221.655,249.939,-61.572,-176.935,6.467,148.274
C03275=1221.650,250.187,-61.599,-176.932,6.469,148.274
C03276=1221.646,250.436,-61.626,-176.929,6.472,148.274
C03277=1221.641,250.685,-61.652,-176.927,6.474,148.274
C03278=1221.636,250.933,-61.679,-176.924,6.476,148.273
C03279=1221.633,251.181,-61.706,-176.922,6.478,148.273
C03280=1221.628,251.430,-61.733,-176.919,6.480,148.273
C03281=1221.624,251.679,-61.758,-176.917,6.482,148.273
C03282=1221.619,251.927,-61.786,-176.915,6.484,148.272
C03283=1221.615,252.175,-61.812,-176.912,6.486,148.272
C03284=1221.610,252.424,-61.838,-176.910,6.488,148.272
C03285=1221.605,252.673,-61.865,-176.907,6.490,148.272
C03286=1221.602,252.921,-61.892,-176.904,6.492,148.271
C03287=1221.597,253.170,-61.919,-176.902,6.495,148.271
C03288=1221.592,253.418,-61.946,-176.899,6.496,148.271
C03289=1221.588,253.667,-61.972,-176.897,6.498,148.271
C03290=1221.583,253.915,-61.999,-176.894,6.500,148.271
C03291=1221.579,254.164,-62.026,-176.892,6.502,148.270
C03292=1221.575,254.412,-62.052,-176.889,6.504,148.270
C03293=1221.570,254.661,-62.079,-176.887,6.506,148.270
C03294=1221.565,254.910,-62.106,-176.885,6.508,148.270
C03295=1221.561,255.158,-62.132,-176.881,6.511,148.269
C03296=1221.557,255.406,-62.159,-176.879,6.513,148.269
C03297=1221.552,255.655,-62.186,-176.877,6.515,148.269
C03298=1221.548,255.903,-62.213,-176.874,6.517,148.269
C03299=1221.543,256.152,-62.240,-176.872,6.519,148.269
C03300=1221.539,256.401,-62.267,-176.869,6.521,148.268
C03301=1221.535,256.649,-62.294,-176.867,6.523,148.268
C03302=1221.531,256.897,-62.321,-176.865,6.525,148.268
C03303=1221.526,257.146,-62.348,-176.861,6.528,148.268
C03304=1221.521,257.394,-62.375,-176.859,6.530,148.268
C03305=1221.517,257.643,-62.402,-176.857,6.532,148.267
C03306=1221.513,257.891,-62.428,-176.854,6.534,148.267
C03307=1221.508,258.140,-62.456,-176.852,6.536,148.267
C03308=1221.504,258.388,-62.483,-176.849,6.538,148.267
C03309=1221.499,258.637,-62.510,-176.847,6.540,148.266
C03310=1221.496,258.886,-62.536,-176.845,6.542,148.266
C03311=1221.491,259.134,-62.564,-176.841,6.545,148.266
C03312=1221.486,259.383,-62.591,-176.839,6.547,148.266
C03313=1221.482,259.631,-62.618,-176.837,6.549,148.266
C03314=1221.477,259.880,-62.645,-176.834,6.551,148.265
C03315=1221.472,260.128,-62.672,-176.832,6.553,148.265
C03316=1221.468,260.376,-62.698,-176.829,6.555,148.265
C03317=1221.464,260.625,-62.726,-176.827,6.557,148.265
C03318=1221.460,260.874,-62.753,-176.824,6.560,148.264
C03319=1221.455,261.122,-62.780,-176.821,6.561,148.264
C03320=1221.451,261.370,-62.808,-176.819,6.564,148.264
C03321=1221.446,261.619,-62.835,-176.817,6.566,148.264
C03322=1221.441,261.867,-62.862,-176.814,6.567,148.264
C03323=1221.437,262.116,-62.889,-176.812,6.570,148.263
C03324=1221.433,262.365,-62.916,-176.809,6.572,148.263
C03325=1221.429,262.612,-62.943,-176.807,6.575,148.263
C03326=1221.424,262.861,-62.970,-176.804,6.576,148.263
C03327=1221.419,263.134,-63.001,-176.801,6.578,148.262
C03328=1221.414,263.407,-63.030,-176.799,6.581,148.262
C03329=1221.410,263.680,-63.060,-176.796,6.583,148.262
C03330=1221.405,263.952,-63.090,-176.793,6.586,148.262
C03331=1221.400,264.201,-63.117,-176.791,6.588,148.262
C03332=1221.396,264.449,-63.145,-176.788,6.590,148.262
C03333=1221.391,264.697,-63.172,-176.786,6.592,148.261
C03334=1221.387,264.946,-63.199,-176.783,6.595,148.261
C03335=1221.383,265.194,-63.227,-176.780,6.597,148.261
C03336=1221.378,265.443,-63.254,-176.778,6.599,148.261
C03337=1221.374,265.691,-63.281,-176.776,6.601,148.261
C03338=1221.370,265.940,-63.309,-176.773,6.603,148.260
C03339=1221.365,266.188,-63.337,-176.771,6.605,148.260
C03340=1221.361,266.437,-63.364,-176.768,6.608,148.260
C03341=1221.356,266.685,-63.391,-176.766,6.610,148.260
C03342=1221.352,266.934,-63.419,-176.763,6.612,148.259
C03343=1221.348,267.182,-63.447,-176.761,6.614,148.259
C03344=1221.343,267.430,-63.474,-176.758,6.616,148.259
C03345=1221.339,267.678,-63.501,-176.756,6.619,148.259
C03346=1221.334,267.928,-63.529,-176.753,6.621,148.259
C03347=1221.329,268.176,-63.557,-176.751,6.623,148.259
C03348=1221.325,268.424,-63.584,-176.748,6.625,148.258
C03349=1221.321,268.673,-63.612,-176.746,6.627,148.258
C03350=1221.317,268.921,-63.640,-176.743,6.630,148.258
C03351=1221.312,269.169,-63.667,-176.741,6.632,148.258
C03352=1221.308,269.418,-63.695,-176.738,6.634,148.258
C03353=1221.304,269.667,-63.722,-176.736,6.636,148.258
C03354=1221.299,269.914,-63.750,-176.733,6.638,148.257
C03355=1221.295,270.163,-63.778,-176.731,6.641,148.257
C03356=1221.290,270.412,-63.805,-176.728,6.643,148.257
C03357=1221.286,270.660,-63.833,-176.726,6.645,148.257
C03358=1221.282,270.909,-63.861,-176.723,6.647,148.257
C03359=1221.277,271.157,-63.888,-176.721,6.650,148.257
C03360=1221.273,271.405,-63.915,-176.718,6.652,148.256
C03361=1221.268,271.654,-63.944,-176.716,6.654,148.256
C03362=1221.264,271.902,-63.972,-176.713,6.656,148.256
C03363=1221.259,272.150,-63.999,-176.711,6.658,148.256
C03364=1221.255,272.399,-64.027,-176.708,6.661,148.256
C03365=1221.251,272.647,-64.055,-176.706,6.663,148.256
C03366=1221.246,272.896,-64.083,-176.703,6.665,148.255
C03367=1221.242,273.144,-64.111,-176.701,6.667,148.255
C03368=1221.238,273.392,-64.138,-176.698,6.670,148.255
C03369=1221.234,273.641,-64.166,-176.696,6.672,148.255
C03370=1221.228,273.890,-64.194,-176.693,6.674,148.255
C03371=1221.224,274.137,-64.222,-176.691,6.676,148.254
C03372=1221.220,274.386,-64.250,-176.688,6.679,148.254
C03373=1221.216,274.635,-64.277,-176.686,6.681,148.254
C03374=1221.211,274.883,-64.306,-176.683,6.683,148.254
C03375=1221.207,275.131,-64.334,-176.681,6.685,148.254
C03376=1221.202,275.379,-64.362,-176.679,6.687,148.253
C03377=1221.198,275.628,-64.390,-176.676,6.690,148.253
C03378=1221.193,275.877,-64.417,-176.674,6.692,148.253
C03379=1221.190,276.125,-64.445,-176.671,6.694,148.253
C03380=1221.184,276.373,-64.474,-176.669,6.696,148.253
C03381=1221.181,276.622,-64.502,-176.666,6.699,148.253
C03382=1221.176,276.870,-64.530,-176.664,6.701,148.253
C03383=1221.172,277.119,-64.559,-176.661,6.703,148.252
C03384=1221.168,277.367,-64.586,-176.659,6.705,148.252
C03385=1221.163,277.616,-64.614,-176.657,6.709,148.252
C03386=1221.158,277.864,-64.642,-176.654,6.710,148.252
C03387=1221.154,278.112,-64.670,-176.652,6.713,148.252
C03388=1221.150,278.360,-64.698,-176.649,6.715,148.252
C03389=1221.145,278.609,-64.726,-176.647,6.718,148.252
C03390=1221.141,278.857,-64.755,-176.644,6.719,148.251
C03391=1221.136,279.105,-64.783,-176.642,6.722,148.251
C03392=1221.133,279.354,-64.811,-176.639,6.725,148.251
C03393=1221.128,279.602,-64.839,-176.637,6.727,148.251
C03394=1221.124,279.851,-64.868,-176.634,6.729,148.251
C03395=1221.119,280.099,-64.895,-176.632,6.731,148.251
C03396=1221.115,280.347,-64.924,-176.629,6.734,148.251
C03397=1221.111,280.595,-64.952,-176.627,6.736,148.251
C03398=1221.106,280.844,-64.981,-176.624,6.738,148.250
C03399=1221.102,281.093,-65.009,-176.622,6.740,148.250
C03400=1221.097,281.341,-65.037,-176.619,6.743,148.250
C03401=1221.094,281.590,-65.065,-176.617,6.745,148.250
C03402=1221.088,281.838,-65.094,-176.615,6.747,148.250
C03403=1221.085,282.086,-65.122,-176.612,6.750,148.250
C03404=1221.080,282.334,-65.151,-176.610,6.752,148.249
C03405=1221.076,282.582,-65.179,-176.608,6.754,148.249
C03406=1221.071,282.831,-65.207,-176.605,6.756,148.249
C03407=1221.067,283.079,-65.235,-176.602,6.759,148.249
C03408=1221.063,283.328,-65.264,-176.600,6.761,148.249
C03409=1221.058,283.576,-65.292,-176.598,6.763,148.249
C03410=1221.054,283.824,-65.321,-176.595,6.766,148.249
C03411=1221.050,284.072,-65.349,-176.592,6.768,148.248
C03412=1221.045,284.321,-65.378,-176.590,6.770,148.248
C03413=1221.040,284.569,-65.406,-176.587,6.774,148.248
C03414=1221.037,284.818,-65.434,-176.585,6.775,148.248
C03415=1221.032,285.066,-65.464,-176.583,6.778,148.248
C03416=1221.028,285.314,-65.492,-176.581,6.780,148.248
C03417=1221.024,285.563,-65.520,-176.577,6.783,148.248
C03418=1221.019,285.811,-65.549,-176.575,6.785,148.248
C03419=1221.015,286.059,-65.578,-176.573,6.787,148.248
C03420=1221.011,286.308,-65.606,-176.570,6.790,148.247
C03421=1221.006,286.556,-65.634,-176.568,6.792,148.247
C03422=1221.002,286.804,-65.664,-176.566,6.794,148.247
C03423=1220.998,287.053,-65.692,-176.563,6.797,148.247
C03424=1220.993,287.301,-65.720,-176.561,6.799,148.247
C03425=1220.989,287.549,-65.750,-176.558,6.801,148.247
C03426=1220.984,287.797,-65.778,-176.556,6.804,148.247
C03427=1220.981,288.045,-65.807,-176.553,6.806,148.246
C03428=1220.976,288.294,-65.836,-176.551,6.808,148.246
C03429=1220.971,288.542,-65.864,-176.549,6.811,148.246
C03430=1220.967,288.790,-65.893,-176.546,6.813,148.246
C03431=1220.962,289.065,-65.925,-176.544,6.816,148.246
C03432=1220.957,289.339,-65.957,-176.541,6.819,148.246
C03433=1220.952,289.614,-65.988,-176.538,6.821,148.246
C03434=1220.948,289.887,-66.021,-176.536,6.824,148.246
C03435=1220.943,290.135,-66.048,-176.533,6.827,148.246
C03436=1220.939,290.383,-66.078,-176.530,6.828,148.245
C03437=1220.935,290.632,-66.107,-176.528,6.831,148.245
C03438=1220.931,290.881,-66.136,-176.526,6.834,148.245
C03439=1220.926,291.128,-66.164,-176.524,6.836,148.245
C03440=1220.922,291.377,-66.193,-176.521,6.838,148.245
C03441=1220.918,291.626,-66.222,-176.518,6.841,148.245
C03442=1220.913,291.873,-66.251,-176.516,6.843,148.245
C03443=1220.908,292.122,-66.280,-176.514,6.845,148.245
C03444=1220.905,292.370,-66.309,-176.511,6.848,148.245
C03445=1220.901,292.618,-66.338,-176.509,6.850,148.245
C03446=1220.896,292.866,-66.367,-176.507,6.852,148.245
C03447=1220.891,293.115,-66.396,-176.504,6.855,148.245
C03448=1220.887,293.364,-66.425,-176.501,6.857,148.244
C03449=1220.883,293.612,-66.454,-176.499,6.860,148.244
C03450=1220.879,293.859,-66.483,-176.497,6.863,148.244
C03451=1220.874,294.108,-66.511,-176.495,6.865,148.244
C03452=1220.870,294.356,-66.541,-176.492,6.868,148.244
C03453=1220.866,294.605,-66.570,-176.489,6.870,148.244
C03454=1220.862,294.853,-66.600,-176.487,6.872,148.244
C03455=1220.857,295.101,-66.628,-176.485,6.875,148.244
C03456=1220.852,295.349,-66.658,-176.482,6.877,148.244
C03457=1220.848,295.598,-66.687,-176.480,6.879,148.244
C03458=1220.844,295.846,-66.716,-176.477,6.882,148.243
C03459=1220.840,296.094,-66.745,-176.475,6.884,148.243
C03460=1220.836,296.342,-66.774,-176.473,6.887,148.243
C03461=1220.831,296.590,-66.803,-176.470,6.890,148.243
C03462=1220.827,296.838,-66.833,-176.468,6.892,148.243
C03463=1220.823,297.087,-66.861,-176.466,6.894,148.243
C03464=1220.818,297.336,-66.891,-176.463,6.897,148.243
C03465=1220.814,297.583,-66.920,-176.461,6.899,148.243
C03466=1220.810,297.831,-66.949,-176.458,6.902,148.243
C03467=1220.805,298.080,-66.979,-176.456,6.904,148.243
C03468=1220.801,298.328,-67.008,-176.454,6.906,148.243
C03469=1220.797,298.577,-67.037,-176.451,6.910,148.243
C03470=1220.793,298.825,-67.067,-176.449,6.912,148.243
C03471=1220.788,299.073,-67.096,-176.446,6.914,148.242
C03472=1220.784,299.321,-67.125,-176.444,6.917,148.242
C03473=1220.779,299.569,-67.155,-176.442,6.919,148.242
C03474=1220.775,299.818,-67.184,-176.440,6.921,148.242
C03475=1220.771,300.066,-67.213,-176.437,6.924,148.242
C03476=1220.767,300.314,-67.243,-176.435,6.926,148.242
C03477=1220.763,300.562,-67.272,-176.432,6.929,148.242
C03478=1220.758,300.811,-67.302,-176.430,6.932,148.242
C03479=1220.754,301.059,-67.332,-176.428,6.934,148.242
C03480=1220.749,301.307,-67.361,-176.425,6.937,148.242
C03481=1220.745,301.555,-67.390,-176.423,6.939,148.242
C03482=1220.740,301.803,-67.420,-176.421,6.941,148.242
C03483=1220.736,302.052,-67.449,-176.418,6.944,148.242
C03484=1220.732,302.300,-67.479,-176.416,6.946,148.242
C03485=1220.728,302.548,-67.508,-176.413,6.949,148.242
C03486=1220.724,302.796,-67.538,-176.411,6.951,148.242
C03487=1220.719,303.045,-67.568,-176.409,6.954,148.241
C03488=1220.715,303.293,-67.597,-176.406,6.957,148.241
C03489=1220.710,303.541,-67.627,-176.404,6.959,148.241
C03490=1220.707,303.789,-67.657,-176.401,6.962,148.241
C03491=1220.702,304.037,-67.686,-176.399,6.964,148.241
C03492=1220.698,304.286,-67.716,-176.397,6.966,148.241
C03493=1220.693,304.534,-67.746,-176.395,6.969,148.241
C03494=1220.689,304.782,-67.775,-176.392,6.972,148.241
C03495=1220.684,305.030,-67.804,-176.390,6.975,148.241
C03496=1220.680,305.278,-67.834,-176.388,6.977,148.241
C03497=1220.676,305.526,-67.864,-176.385,6.979,148.241
C03498=1220.671,305.775,-67.894,-176.382,6.982,148.241
C03499=1220.667,306.023,-67.923,-176.380,6.984,148.241
C03500=1220.663,306.271,-67.953,-176.378,6.986,148.241
C03501=1220.659,306.519,-67.983,-176.375,6.989,148.241
C03502=1220.654,306.767,-68.013,-176.373,6.992,148.241
C03503=1220.650,307.016,-68.043,-176.371,6.995,148.241
C03504=1220.646,307.264,-68.072,-176.369,6.997,148.241
C03505=1220.642,307.511,-68.102,-176.366,6.999,148.241
C03506=1220.637,307.760,-68.132,-176.364,7.002,148.241
C03507=1220.633,308.008,-68.162,-176.362,7.005,148.241
C03508=1220.629,308.256,-68.192,-176.360,7.008,148.241
C03509=1220.624,308.505,-68.222,-176.357,7.010,148.241
C03510=1220.620,308.753,-68.251,-176.355,7.012,148.241
C03511=1220.616,309.000,-68.281,-176.353,7.015,148.241
C03512=1220.612,309.250,-68.312,-176.350,7.017,148.241
C03513=1220.608,309.497,-68.342,-176.348,7.020,148.241
C03514=1220.604,309.746,-68.372,-176.346,7.023,148.241
C03515=1220.599,309.994,-68.402,-176.343,7.026,148.241
C03516=1220.595,310.242,-68.432,-176.341,7.028,148.240
C03517=1220.591,310.490,-68.461,-176.339,7.030,148.240
C03518=1220.586,310.738,-68.492,-176.336,7.033,148.240
C03519=1220.582,310.986,-68.521,-176.334,7.035,148.240
C03520=1220.577,311.234,-68.552,-176.331,7.038,148.240
C03521=1220.573,311.483,-68.582,-176.329,7.041,148.240
C03522=1220.569,311.730,-68.612,-176.327,7.043,148.240
C03523=1220.564,311.979,-68.642,-176.325,7.046,148.240
C03524=1220.560,312.226,-68.672,-176.323,7.048,148.240
C03525=1220.555,312.475,-68.702,-176.320,7.051,148.240
C03526=1220.552,312.723,-68.733,-176.318,7.054,148.240
C03527=1220.547,312.972,-68.763,-176.316,7.056,148.240
C03528=1220.543,313.220,-68.793,-176.313,7.059,148.240
C03529=1220.539,313.468,-68.822,-176.311,7.061,148.240
C03530=1220.535,313.716,-68.853,-176.309,7.064,148.240
C03531=1220.531,313.964,-68.883,-176.306,7.066,148.240
C03532=1220.526,314.212,-68.913,-176.304,7.070,148.240
C03533=1220.522,314.460,-68.943,-176.302,7.072,148.240
C03534=1220.518,314.709,-68.974,-176.300,7.074,148.240
C03535=1220.513,314.984,-69.007,-176.297,7.077,148.240
C03536=1220.508,315.260,-69.041,-176.295,7.080,148.240
C03537=1220.503,315.536,-69.075,-176.292,7.083,148.240
C03538=1220.499,315.811,-69.109,-176.289,7.086,148.240
C03539=1220.494,316.060,-69.139,-176.287,7.089,148.240
C03540=1220.489,316.308,-69.169,-176.286,7.091,148.240
C03541=1220.486,316.556,-69.200,-176.283,7.094,148.240
C03542=1220.481,316.805,-69.230,-176.281,7.096,148.240
C03543=1220.477,317.053,-69.260,-176.278,7.099,148.240
C03544=1220.473,317.301,-69.291,-176.276,7.102,148.240
C03545=1220.469,317.548,-69.321,-176.274,7.105,148.241
C03546=1220.465,317.797,-69.352,-176.272,7.107,148.241
C03547=1220.460,318.045,-69.382,-176.270,7.109,148.240
C03548=1220.456,318.293,-69.413,-176.267,7.113,148.240
C03549=1220.451,318.541,-69.443,-176.265,7.115,148.240
C03550=1220.448,318.789,-69.473,-176.263,7.118,148.241
C03551=1220.444,319.037,-69.505,-176.261,7.120,148.241
C03552=1220.439,319.286,-69.535,-176.259,7.123,148.241
C03553=1220.435,319.534,-69.565,-176.256,7.126,148.241
C03554=1220.430,319.782,-69.596,-176.254,7.128,148.241
C03555=1220.426,320.030,-69.627,-176.252,7.131,148.241
C03556=1220.422,320.278,-69.657,-176.249,7.133,148.241
C03557=1220.418,320.526,-69.688,-176.247,7.136,148.241
C03558=1220.413,320.774,-69.718,-176.245,7.139,148.241
C03559=1220.410,321.022,-69.749,-176.243,7.141,148.241
C03560=1220.405,321.270,-69.780,-176.240,7.144,148.241
C03561=1220.401,321.518,-69.810,-176.239,7.147,148.241
C03562=1220.396,321.766,-69.840,-176.236,7.150,148.241
C03563=1220.392,322.015,-69.871,-176.234,7.152,148.241
C03564=1220.388,322.263,-69.902,-176.231,7.155,148.241
C03565=1220.384,322.511,-69.932,-176.230,7.158,148.241
C03566=1220.380,322.759,-69.963,-176.228,7.160,148.241
C03567=1220.375,323.007,-69.994,-176.225,7.163,148.241
C03568=1220.371,323.254,-70.025,-176.223,7.165,148.241
C03569=1220.367,323.502,-70.055,-176.221,7.168,148.241
C03570=1220.363,323.751,-70.087,-176.218,7.171,148.241
C03571=1220.358,323.999,-70.117,-176.216,7.174,148.241
C03572=1220.354,324.247,-70.148,-176.214,7.176,148.241
C03573=1220.351,324.495,-70.179,-176.213,7.179,148.242
C03574=1220.346,324.743,-70.209,-176.210,7.182,148.242
C03575=1220.341,324.991,-70.240,-176.208,7.184,148.241
C03576=1220.337,325.240,-70.271,-176.206,7.187,148.242
C03577=1220.333,325.488,-70.302,-176.203,7.190,148.242
C03578=1220.329,325.735,-70.333,-176.201,7.193,148.242
C03579=1220.325,325.983,-70.364,-176.199,7.195,148.242
C03580=1220.321,326.231,-70.395,-176.197,7.197,148.242
C03581=1220.316,326.479,-70.426,-176.195,7.201,148.242
C03582=1220.312,326.728,-70.457,-176.193,7.203,148.242
C03583=1220.307,326.976,-70.488,-176.190,7.206,148.242
C03584=1220.304,327.224,-70.519,-176.188,7.208,148.242
C03585=1220.300,327.471,-70.550,-176.186,7.212,148.242
C03586=1220.295,327.719,-70.580,-176.184,7.214,148.242
C03587=1220.291,327.968,-70.611,-176.182,7.216,148.242
C03588=1220.287,328.215,-70.643,-176.180,7.220,148.243
C03589=1220.282,328.463,-70.674,-176.178,7.222,148.242
C03590=1220.278,328.712,-70.705,-176.176,7.225,148.243
C03591=1220.274,328.960,-70.736,-176.173,7.227,148.243
C03592=1220.270,329.208,-70.767,-176.171,7.230,148.243
C03593=1220.265,329.456,-70.798,-176.169,7.233,148.243
C03594=1220.261,329.704,-70.829,-176.167,7.235,148.243
C03595=1220.257,329.952,-70.861,-176.165,7.239,148.243
C03596=1220.252,330.200,-70.892,-176.163,7.241,148.243
C03597=1220.249,330.448,-70.922,-176.161,7.244,148.243
C03598=1220.245,330.696,-70.954,-176.158,7.246,148.243
C03599=1220.241,330.944,-70.985,-176.156,7.250,148.243
C03600=1220.236,331.192,-71.016,-176.154,7.252,148.243
C03601=1220.232,331.440,-71.047,-176.153,7.254,148.243
C03602=1220.228,331.688,-71.078,-176.150,7.258,148.244
C03603=1220.223,331.936,-71.110,-176.148,7.260,148.244
C03604=1220.219,332.184,-71.141,-176.146,7.263,148.244
C03605=1220.215,332.432,-71.172,-176.144,7.266,148.244
C03606=1220.211,332.680,-71.203,-176.142,7.269,148.244
C03607=1220.206,332.928,-71.235,-176.140,7.271,148.244
C03608=1220.202,333.177,-71.267,-176.138,7.274,148.244
C03609=1220.198,333.424,-71.298,-176.135,7.277,148.244
C03610=1220.194,333.673,-71.329,-176.134,7.279,148.244
C03611=1220.189,333.920,-71.361,-176.132,7.283,148.245
C03612=1220.185,334.168,-71.391,-176.129,7.285,148.245
C03613=1220.181,334.416,-71.423,-176.128,7.287,148.245
C03614=1220.177,334.664,-71.454,-176.125,7.290,148.245
C03615=1220.173,334.912,-71.486,-176.124,7.293,148.245
C03616=1220.168,335.159,-71.517,-176.121,7.296,148.245
C03617=1220.164,335.408,-71.548,-176.119,7.299,148.245
C03618=1220.160,335.655,-71.580,-176.117,7.302,148.245
C03619=1220.155,335.904,-71.612,-176.115,7.304,148.245
C03620=1220.152,336.152,-71.643,-176.113,7.307,148.245
C03621=1220.147,336.400,-71.675,-176.111,7.310,148.246
C03622=1220.143,336.648,-71.706,-176.109,7.312,148.246
C03623=1220.139,336.896,-71.738,-176.107,7.316,148.246
C03624=1220.135,337.144,-71.769,-176.105,7.318,148.246
C03625=1220.131,337.392,-71.800,-176.103,7.320,148.246
C03626=1220.126,337.640,-71.833,-176.101,7.324,148.246
C03627=1220.122,337.887,-71.864,-176.099,7.326,148.246
C03628=1220.118,338.136,-71.895,-176.097,7.330,148.247
C03629=1220.114,338.383,-71.927,-176.095,7.332,148.247
C03630=1220.110,338.631,-71.959,-176.093,7.334,148.247
C03631=1220.106,338.880,-71.991,-176.091,7.338,148.247
C03632=1220.101,339.128,-72.022,-176.089,7.340,148.247
C03633=1220.097,339.376,-72.054,-176.087,7.343,148.247
C03634=1220.093,339.623,-72.085,-176.085,7.346,148.247
C03635=1220.089,339.871,-72.117,-176.084,7.348,148.248
C03636=1220.084,340.119,-72.148,-176.081,7.351,148.248
C03637=1220.080,340.367,-72.180,-176.079,7.354,148.248
C03638=1220.076,340.615,-72.212,-176.077,7.357,148.248
C03639=1220.071,340.893,-72.248,-176.075,7.361,148.248
C03640=1220.067,341.171,-72.283,-176.073,7.363,148.248
C03641=1220.062,341.449,-72.319,-176.071,7.366,148.248
C03642=1220.057,341.727,-72.355,-176.068,7.370,148.249
C03643=1220.053,341.974,-72.386,-176.067,7.372,148.249
C03644=1220.049,342.222,-72.418,-176.065,7.375,148.249
C03645=1220.044,342.470,-72.450,-176.062,7.378,148.249
C03646=1220.040,342.718,-72.481,-176.060,7.381,148.249
C03647=1220.037,342.966,-72.513,-176.059,7.384,148.249
C03648=1220.032,343.214,-72.545,-176.057,7.386,148.250
C03649=1220.028,343.462,-72.577,-176.055,7.389,148.250
C03650=1220.024,343.710,-72.609,-176.053,7.392,148.250
C03651=1220.019,343.958,-72.641,-176.051,7.394,148.250
